// TwinCAT 3 PLC project x_template_xPlc
// Title: x_template_xPlc
// Company: TcOpen.MTS
// ProjectVersion: 0.6.0.913
// ProgramVersion: 3.1.4023.0
// libraries:
//   Tc2_Standard, * (Beckhoff Automation GmbH)
//   Tc2_System, * (Beckhoff Automation GmbH)
//   Tc3_Module, * (Beckhoff Automation GmbH)
//   TcoAbbRobotics, 0.11.0.74 (Vortex.Library)
//   TcoAbstractions, 0.11.0.74 (Vortex.Library)
//   TcoAimTtiPowerSupply, 0.11.0.74 (Vortex.Library)
//   TcoCognexVision, 0.11.0.74 (Vortex.Library)
//   TcoCore, 0.11.0.74 (Vortex.Library)
//   TcoData, 0.11.0.74 (Vortex.Library)
//   TcoDrivesBeckhoff, 0.11.0.74 (Vortex.Library)
//   TcoElements, 0.11.0.74 (Vortex.Library)
//   TcoInspectors, 0.11.0.74 (Vortex.Library)
//   TcoIo, 0.11.0.74 (Vortex.Library)
//   TcoKukaRobotics, 0.11.0.74 (Vortex.Library)
//   TcoMitsubishiRobotics, 0.11.0.74 (Vortex.Library)
//   TcoPneumatics, 0.11.0.74 (Vortex.Library)
//   TcoRexrothPress, 0.11.0.74 (Vortex.Library)
//   TcoTixonFeeding, 0.11.0.74 (Vortex.Library)
//   TcoUrRobotics, 0.11.0.74 (Vortex.Library)
//   TcoUtilities, 0.11.0.74 (Vortex.Library)
// project tree:
//   Abstractions/Components/ArrayRenderingExample/ SampleArrayToRender.TcDUT, SampleDataItem.TcDUT
//   Abstractions/Components/MtsFeeding/Blisters/Plb/ TcoPlbPaletizator.TcPOU, TcoPlbPaletizator_Components.TcDUT, TcoPlbPaletizator_Config_v_1_x_x.TcDUT, TcoPlbPaletizator_Control_v_1_x_x.TcDUT, TcoPlbPaletizator_Positions.TcPOU, TcoPlbPaletizator_Status_v_1_x_x.TcDUT
//   Abstractions/Components/MtsFeeding/Blisters/Plr/ TcoPlrPaletizator.TcPOU, TcoPlrPaletizator_Components.TcDUT, TcoPlrPaletizator_Config_v_1_x_x.TcDUT, TcoPlrPaletizator_Control_v_1_x_x.TcDUT, TcoPlrPaletizator_Status_v_1_x_x.TcDUT
//   Abstractions/Components/MtsFeeding/Blisters/Pls/ TcoPlsPaletizator.TcPOU, TcoPlsPaletizator_Components.TcDUT, TcoPlsPaletizator_Config_v_1_x_x.TcDUT, TcoPlsPaletizator_Control_v_1_x_x.TcDUT, TcoPlsPaletizator_Status_v_1_x_x.TcDUT
//   Abstractions/Components/MtsFeeding/Blisters/ TcoFeeding_Config_v_1_x_x.TcDUT, TcoFeeding_Status_v_1_x_x.TcDUT
//   Abstractions/Components/MtsFeeding/Components/OscilatingConveyorFeeder/ eTcoOscilatingConveyorOscilationModes.TcDUT, eTcoOscilatingConveyorStatus.TcDUT, TcoOscilatingConveyorFeeder.TcPOU, TcoOscilatingConveyorFeederComponents.TcDUT, TcoOscilatingConveyorFeeder_Config_v_1_x_x.TcDUT, TcoOscilatingConveyorFeeder_Control_v_1_x_x.TcDUT, TcoOscilatingConveyorFeeder_DesignerSpecificData.TcPOU, TcoOscilatingConveyorFeeder_PcToPlc.TcDUT, TcoOscilatingConveyorFeeder_PlcToPc.TcDUT, TcoOscilatingConveyorFeeder_Status_v_1_x_x.TcDUT
//   Abstractions/Components/MtsFeeding/ TcoFeedingSequenceTask.TcPOU
//   Abstractions/Components/Rework/ eReworkResults.TcDUT, ReworkData.TcDUT, ReworkInstructionTask.TcPOU
//   Abstractions/Components/TS/EqTransfer/ eTcoEq2TransferConfiguration.TcDUT, eTcoEq2TransferHandlingMode.TcDUT, TcoEq2Transfer.TcPOU, TcoEq2TransferComponents.TcDUT, TcoEq2Transfer_Config.TcDUT, TcoEq2Transfer_Control.TcDUT, TcoEq2Transfer_Status.TcDUT
//   Abstractions/Components/TS/RotaryTrabsferWithLift/ TcoLiftingRotaryTransfer.TcPOU, TcoLiftingRotaryTransferComponents.TcDUT, TcoLiftingRotaryTransfer_Config.TcDUT, TcoLiftingRotaryTransfer_Control.TcDUT, TcoLiftingRotaryTransfer_Status.TcDUT
//   Abstractions/Components/TS/RotaryTransfer/ TcoRotaryTransfer.TcPOU, TcoRotaryTransferComponents.TcDUT, TcoRotaryTransfer_Config.TcDUT, TcoRotaryTransfer_Control.TcDUT, TcoRotaryTransfer_Status.TcDUT
//   Abstractions/Components/TS/WorkPosition/ TcoTransferSystemComponent.TcPOU, TcoTransferSystemComponents.TcDUT, TcoTransferSystem_Config.TcDUT, TcoTransferSystem_Control.TcDUT, TcoTransferSystem_Status.TcDUT
//   Abstractions/Components/WrappedComponent/ WrappedComponentExample.TcPOU, WrappedComponentExample_Config.TcDUT, WrappedComponentExample_Control.TcDUT, WrappedComponentExample_Status.TcDUT, WrappedComponentsExample.TcDUT
//   Abstractions/CUBase/ CuBaseRecurringFail.TcDUT, CuBaseRecurringFailures.TcDUT, CUBase.TcPOU, CUBaseStatusInfo.TcDUT, CUBaseSettings.TcDUT, CUComponentsBase.TcDUT (not stored), ICUBase.TcIO, ICUTask.TcIO (not stored), OperatorInfo.TcDUT (not stored)
//   Abstractions/CUBase/Data/ BasicCounterData.TcDUT, CuHeader.TcDUT, CUProcessDataBase.TcDUT, CUTechnologicalDataBase.TcDUT, eCUMode.TcDUT (not stored), eCUState.TcDUT, eDataEntityInvokeType.TcDUT, EntityHeader.TcDUT
//   Abstractions/CUBase/RemoteTasks/ ProductionPlaner.TcPOU
//   Abstractions/CUBase/Tasks/ CUBaseAutomat.TcPOU, CUBaseSuspend.TcPOU, CUBaseGround.TcPOU (not stored), CUBaseRecover.TcPOU
//   Abstractions/Generic/LightTower/ TcoLightTower.TcPOU, TcoLightTower_Config.TcDUT, TcoLightTower_Info.TcDUT, TcoLightTower_Status.TcDUT
//   Abstractions/Generic/NotificationPanel/ NotificationPanel.TcPOU, NotificationPanelInfo.TcDUT
//   Abstractions/Generic/TagsPairing/ eTagPairingAnswer.TcDUT, eTagPairingMode.TcDUT, eTagPairingStatus.TcDUT, PairTagTask.TcPOU, TagsPairing.TcDUT
//   Abstractions/Safety/ControlButtons/ ITcoControlButtons.TcIO, TcoControlButtons.TcPOU, TcoControledZone_Info.TcDUT
//   Abstractions/Safety/ControlledZone/ TcoControlledZone.TcPOU, TcoControlledZoneActionTask.TcPOU, TcoControlledZone_Config.TcDUT, TcoControlledZone_Status.TcDUT
//   Abstractions/Safety/ControlVoltage/ ITcoControlVoltage.TcIO, TcoControlVoltage.TcPOU
//   Abstractions/Safety/DoorCircuit/ TcoDoorCircuit_Status.TcDUT, TcoDoorCircuit_Config.TcDUT, TcoDoorCircuit.TcPOU, ITcoDoorCircuit.TcIO
//   Abstractions/Safety/Doors/ ITcoDoorLock.TcIO (not stored), TcoStandardDoor.TcPOU, TcoBasicDoor.TcPOU
//   Abstractions/Safety/Estop/ TcoEmergencyStop.TcPOU
//   Abstractions/Safety/KeyMode/ TcoKeyMode_Config.TcDUT, TcoKeyMode_Status.TcDUT, TcoKeyMode.TcPOU, ITcoKeyMode.TcIO
//   Abstractions/Safety/KeyNormalService/ TcoKeyNormalService.TcPOU, ITcoKeyNormalSevice.TcIO
//   Abstractions/TcoCore/ CycleTimeAnalitics.TcDUT, TcoInnerTask.TcPOU (not stored), TcoTaskedSequencer.TcPOU, TcoTaskedService.TcPOU (not stored)
//   Abstractions/Technology/ eStations.TcDUT (not stored)
//   DUTs/IO_Specific/Aventics/ AES_D_BC_ECAT_Gen2_32bytes_Data_Inputs.TcDUT, AES_D_BC_ECAT_Gen2_32bytes_Data_Outputs.TcDUT, AES_D_BC_ECAT_Gen2_4bytes_Data_Inputs.TcDUT, AES_D_BC_ECAT_Gen2_4bytes_Data_Outputs.TcDUT
//   / MAIN.TcPOU (not stored), PlcTask.TcTTO
//   Technology/CU00x/Automat/ CU00xAutomatParalell_1_Task.TcPOU, CU00xAutomatTask.TcPOU
//   Technology/CU00x/Components/ CU00xExamplesOfComponents.TcDUT, CU00xComponents.TcDUT
//   Technology/CU00x/Data/ CU00xTechnologicalData.TcDUT, CU00xDialogContent.TcPOU, CU00xProcessData.TcDUT
//   Technology/CU00x/Ground/ CU00xGroundTask.TcPOU
//   Technology/CU00x/Manual/ CU00xManualTask.TcPOU
//   Technology/CU00x/Positions/ CU00xTestMultiPositions.TcPOU, Cu00xTestPositions.TcPOU
//   Technology/CU00x/Safety/Suspend/ CU00xSuspendTask.TcPOU
//   Technology/CU00x/Safety/Recover/ CU00xRecoverTask.TcPOU
//   Technology/Data/ InternalStorage.TcPOU, ProcessData.TcDUT, ProcessDataManager.TcPOU, TcoEntityBase.TcDUT, TechnologicalDataManager.TcPOU (not stored), TechnologyData.TcDUT
//   Technology/CU00x/ CU00x.TcPOU
//   Technology/ Technology.TcPOU, TechnologyComponents.TcDUT
//   DUTs/IO/PDOs/ Device_State_F0482DC3.TcDUT (not stored), Device_Control_6258066A.TcDUT (not stored), Inputs_23559BB0.TcDUT (not stored), Outputs_FC2FACAD.TcDUT (not stored), Modules_85784B27.TcDUT (not stored), Channel_830843C1.TcDUT, Channel_42CA91F7.TcDUT
//   DUTs/IO/Boxes/ EK1200_013D0B49.TcDUT, EK1122_1FC0878B.TcDUT, AES_510494FB.TcDUT (not stored), EPP1322_1FC0878B.TcDUT (not stored), EPP1809_32157CFD.TcDUT (not stored), EPP1008_78E8D3DD.TcDUT (not stored), EL1809_32157CFD.TcDUT, EL2809_2B6483BD.TcDUT, EL9011_D65D3D32.TcDUT
//   DUTs/IO/Devices/ SyncUnitTasks_4BE01469.TcDUT, SyncUnits_67D36DDA.TcDUT
//   DUTs/IO/Topology/ EK_E812B8FA.TcDUT (not stored), EC_4E5C738F.TcDUT (not stored), EC_245FBB9A.TcDUT (not stored)
//   GVLs/ GVL_iXlinker.TcGVL
// real-time tasks:
//   TASK PlcTask: cycle T#10ms, priority 20, ADS port 350
//   TASK PlcTask1: cycle T#10ms, priority 21, ADS port 351
// I/O:
//   DEVICE EC1 (disabled), AmsNetId 192.168.4.1.7.1
//     (EK1200) [EK1200-5000 EtherCAT Power supply (2A E-Bus)]
//       EC (EK1122) [EK1122 2 port EtherCAT junction]
//       PN (EL6631) [EL6631 PROFINET IO Controller]
//       IA1 (EL1809) [EL1809 16Ch. Dig. Input 24V, 3ms]
//       QA1 (EL2809) [EL2809 16Ch. Dig. Output 24V, 0.5A]
//       Term 6 (EL4004) [EL4004 4Ch. Ana. Output 0-10V, 12bit]
//       Term 7 (EL7342) [EL7342 2Ch. DC motor output stage (50V, 3.5A)]
//       Term 8 (EL4004) [EL4004 4Ch. Ana. Output 0-10V, 12bit]
//       Term 9 (EL6001) [EL6001 Interface (RS232)]
//       Term 13 (EL9011) [EL9011 End Terminal]
//   DEVICE EC (disabled), AmsNetId 192.168.4.1.2.1
//     EC [EK1200-5000 EtherCAT Power supply (2A E-Bus)]
//       EK [EK1122 2 port EtherCAT junction]
//         PNEU [AES Fieldbus Coupler Gen2]
//           modules: Modules
//         AB [EPP1322-0001 3 port EtherCAT P gateway]
//         AB21 [EPP1809-0021 16 Ch. Dig. Input 24V, 3ms, M8]
//         AB22 [EPP1809-0021 16 Ch. Dig. Input 24V, 3ms, M8]
//         AB23 [EPP1008-0001 8 Ch. Dig. Input 24V, 3ms, M8]
//         AB24 [EPP1008-0001 8 Ch. Dig. Input 24V, 3ms, M8]
//       IA1 [EL1809 16Ch. Dig. Input 24V, 3ms]
//       QA1 [EL2809-0015 16Ch. Dig. Output 24V DC, 0.35A, not short-circuit proof]
//       Term 11 (EL9011) [EL9011 End Terminal]
// variable links:
//   x_template_xPlc/x_template_xPlc Instance <-> EC
//     PlcTask Inputs/GVL_iXlinker.EC.InfoData.AmsNetId <-> InfoData/AmsNetId
//     PlcTask Inputs/GVL_iXlinker.EC.InfoData.CfgSlaveCount <-> InfoData/CfgSlaveCount
//     PlcTask Inputs/GVL_iXlinker.EC.InfoData.ChangeCount <-> InfoData/ChangeCount
//     PlcTask Inputs/GVL_iXlinker.EC.InfoData.DevId <-> InfoData/DevId
//     PlcTask Inputs/GVL_iXlinker.EC.Inputs.DevState <-> Inputs/DevState
//     PlcTask Inputs/GVL_iXlinker.EC.Inputs.Frm0InputToggle <-> Inputs/Frm0InputToggle
//     PlcTask Inputs/GVL_iXlinker.EC.Inputs.Frm0State <-> Inputs/Frm0State
//     PlcTask Inputs/GVL_iXlinker.EC.Inputs.Frm0WcState <-> Inputs/Frm0WcState
//     PlcTask Inputs/GVL_iXlinker.EC.Inputs.SlaveCount <-> Inputs/SlaveCount
//     PlcTask Inputs/GVL_iXlinker.EC.SyncUnits._default.PlcTask.InfoData.ObjectId <-> SyncUnits/<default>/PlcTask/InfoData/ObjectId
//     PlcTask Inputs/GVL_iXlinker.EC.SyncUnits._default.PlcTask.InfoData.SlaveCount <-> SyncUnits/<default>/PlcTask/InfoData/SlaveCount
//     PlcTask Inputs/GVL_iXlinker.EC.SyncUnits._default.PlcTask.InfoData.State <-> SyncUnits/<default>/PlcTask/InfoData/State
//     PlcTask Inputs/GVL_iXlinker.EC.SyncUnits._default.PlcTask.WcState.WcState <-> SyncUnits/<default>/PlcTask/WcState/WcState
//     PlcTask Outputs/GVL_iXlinker.EC.Outputs.DevCtrl <-> Outputs/DevCtrl
//     PlcTask Outputs/GVL_iXlinker.EC.Outputs.Frm0Ctrl <-> Outputs/Frm0Ctrl
//     PlcTask Outputs/GVL_iXlinker.EC.Outputs.Frm0WcCtrl <-> Outputs/Frm0WcCtrl
//   x_template_xPlc/x_template_xPlc Instance <-> EC/EC/EK
//     PlcTask Inputs/GVL_iXlinker.EC.EC.EK.InfoData.State <-> InfoData/State
//   x_template_xPlc/x_template_xPlc Instance <-> EC/EC/EK/AB
//     PlcTask Inputs/GVL_iXlinker.EC.EC.EK.AB.InfoData.State <-> InfoData/State
//   x_template_xPlc/x_template_xPlc Instance <-> EC/EC/EK/AB21
//     PlcTask Inputs/GVL_iXlinker.EC.EC.EK.AB21.Channel_{1..16}.Input <-> Channel {1..16}/Input  (16 links)
//     PlcTask Inputs/GVL_iXlinker.EC.EC.EK.AB21.InfoData.State <-> InfoData/State
//     PlcTask Inputs/GVL_iXlinker.EC.EC.EK.AB21.WcState.InputToggle <-> WcState/InputToggle
//     PlcTask Inputs/GVL_iXlinker.EC.EC.EK.AB21.WcState.WcState <-> WcState/WcState
//   x_template_xPlc/x_template_xPlc Instance <-> EC/EC/EK/AB22
//     PlcTask Inputs/GVL_iXlinker.EC.EC.EK.AB22.Channel_{1..16}.Input <-> Channel {1..16}/Input  (16 links)
//     PlcTask Inputs/GVL_iXlinker.EC.EC.EK.AB22.InfoData.State <-> InfoData/State
//     PlcTask Inputs/GVL_iXlinker.EC.EC.EK.AB22.WcState.InputToggle <-> WcState/InputToggle
//     PlcTask Inputs/GVL_iXlinker.EC.EC.EK.AB22.WcState.WcState <-> WcState/WcState
//   x_template_xPlc/x_template_xPlc Instance <-> EC/EC/EK/AB23
//     PlcTask Inputs/GVL_iXlinker.EC.EC.EK.AB23.Channel_{1..8}.Input <-> Channel {1..8}/Input  (8 links)
//     PlcTask Inputs/GVL_iXlinker.EC.EC.EK.AB23.InfoData.State <-> InfoData/State
//     PlcTask Inputs/GVL_iXlinker.EC.EC.EK.AB23.WcState.InputToggle <-> WcState/InputToggle
//     PlcTask Inputs/GVL_iXlinker.EC.EC.EK.AB23.WcState.WcState <-> WcState/WcState
//   x_template_xPlc/x_template_xPlc Instance <-> EC/EC/EK/AB24
//     PlcTask Inputs/GVL_iXlinker.EC.EC.EK.AB24.Channel_{1..8}.Input <-> Channel {1..8}/Input  (8 links)
//     PlcTask Inputs/GVL_iXlinker.EC.EC.EK.AB24.InfoData.State <-> InfoData/State
//     PlcTask Inputs/GVL_iXlinker.EC.EC.EK.AB24.WcState.InputToggle <-> WcState/InputToggle
//     PlcTask Inputs/GVL_iXlinker.EC.EC.EK.AB24.WcState.WcState <-> WcState/WcState
//   x_template_xPlc/x_template_xPlc Instance <-> EC/EC/EK/PNEU
//     PlcTask Inputs/GVL_iXlinker.EC.EC.EK.PNEU.Device_State.CommonValve <-> Device_State/CommonValve
//     PlcTask Inputs/GVL_iXlinker.EC.EC.EK.PNEU.Device_State.Configuration_Error_IO_Module <-> Device_State/Configuration Error IO-Module
//     PlcTask Inputs/GVL_iXlinker.EC.EC.EK.PNEU.Device_State.Configuration_Error_Valve <-> Device_State/Configuration Error Valve
//     PlcTask Inputs/GVL_iXlinker.EC.EC.EK.PNEU.Device_State.Configuratipn_Error_SLS <-> Device_State/Configuratipn Error SLS
//     PlcTask Inputs/GVL_iXlinker.EC.EC.EK.PNEU.Device_State.Count_IO_Module_to_big <-> Device_State/Count IO-Module to big
//     PlcTask Inputs/GVL_iXlinker.EC.EC.EK.PNEU.Device_State.Heardbeat_x <-> Device_State/Heardbeat
//     PlcTask Inputs/GVL_iXlinker.EC.EC.EK.PNEU.Device_State.IO_1_8 <-> Device_State/IO:1-8
//     PlcTask Inputs/GVL_iXlinker.EC.EC.EK.PNEU.Device_State.IO_9_10 <-> Device_State/IO:9-10
//     PlcTask Inputs/GVL_iXlinker.EC.EC.EK.PNEU.Device_State.Switchcounter_Error <-> Device_State/Switchcounter Error
//     PlcTask Inputs/GVL_iXlinker.EC.EC.EK.PNEU.Device_State.UA_OFF <-> Device_State/UA OFF
//     PlcTask Inputs/GVL_iXlinker.EC.EC.EK.PNEU.Device_State.UL_OFF <-> Device_State/UL OFF
//     PlcTask Inputs/GVL_iXlinker.EC.EC.EK.PNEU.Device_State.Undervoltage_5V <-> Device_State/Undervoltage 5V
//     PlcTask Inputs/GVL_iXlinker.EC.EC.EK.PNEU.Device_State.Undervoltage_UA <-> Device_State/Undervoltage UA
//     PlcTask Inputs/GVL_iXlinker.EC.EC.EK.PNEU.Device_State.Undervoltage_UL <-> Device_State/Undervoltage UL
//     PlcTask Inputs/GVL_iXlinker.EC.EC.EK.PNEU.Device_State.Unknown_Module_ID <-> Device_State/Unknown Module ID
//     PlcTask Inputs/GVL_iXlinker.EC.EC.EK.PNEU.Device_State.ValveExtSupplyDiag_1_6 <-> Device_State/ValveExtSupplyDiag:1-6
//     PlcTask Inputs/GVL_iXlinker.EC.EC.EK.PNEU.InfoData.AdsAddr <-> InfoData/AdsAddr
//     PlcTask Inputs/GVL_iXlinker.EC.EC.EK.PNEU.InfoData.State <-> InfoData/State
//     PlcTask Inputs/GVL_iXlinker.EC.EC.EK.PNEU.Modules.Inputs.digital_Data_I[{0..31}] <-> Modules/Inputs/digital Data I_{0..31}  (32 links)
//     PlcTask Inputs/GVL_iXlinker.EC.EC.EK.PNEU.WcState.InputToggle <-> WcState/InputToggle
//     PlcTask Inputs/GVL_iXlinker.EC.EC.EK.PNEU.WcState.WcState <-> WcState/WcState
//     PlcTask Outputs/GVL_iXlinker.EC.EC.EK.PNEU.Device_Control.Default_Modul_Control <-> Device_Control/Default_Modul_Control
//     PlcTask Outputs/GVL_iXlinker.EC.EC.EK.PNEU.Device_Control.Freeze_Output <-> Device_Control/Freeze Output
//     PlcTask Outputs/GVL_iXlinker.EC.EC.EK.PNEU.Device_Control.HL_Swap <-> Device_Control/HL_Swap
//     PlcTask Outputs/GVL_iXlinker.EC.EC.EK.PNEU.Device_Control.Web_App_Disable <-> Device_Control/Web App Disable
//     PlcTask Outputs/GVL_iXlinker.EC.EC.EK.PNEU.Modules.Outputs.digital_Data_O[{0..31}] <-> Modules/Outputs/digital Data O_{0..31}  (32 links)
//   x_template_xPlc/x_template_xPlc Instance <-> EC/EC/IA1
//     PlcTask Inputs/GVL_iXlinker.EC.EC.IA1.Channel_{1..16}.Input <-> Channel {1..16}/Input  (16 links)
//     PlcTask Inputs/GVL_iXlinker.EC.EC.IA1.InfoData.State <-> InfoData/State
//     PlcTask Inputs/GVL_iXlinker.EC.EC.IA1.WcState.InputToggle <-> WcState/InputToggle
//     PlcTask Inputs/GVL_iXlinker.EC.EC.IA1.WcState.WcState <-> WcState/WcState
//   x_template_xPlc/x_template_xPlc Instance <-> EC/EC/QA1
//     PlcTask Inputs/GVL_iXlinker.EC.EC.QA1.InfoData.State <-> InfoData/State
//     PlcTask Inputs/GVL_iXlinker.EC.EC.QA1.WcState.WcState <-> WcState/WcState
//     PlcTask Outputs/GVL_iXlinker.EC.EC.QA1.Channel_{1..16}.Output <-> Channel {1..16}/Output  (16 links)

CONFIGURATION x_template_xPlc
    RESOURCE PLC ON TwinCAT3
        TASK PlcTask(INTERVAL := T#4ms, PRIORITY := 20);
        PROGRAM MAIN WITH PlcTask : MAIN;
    END_RESOURCE
END_CONFIGURATION

// ---- Abstractions/Components/ArrayRenderingExample/SampleArrayToRender.TcDUT
TYPE SampleArrayToRender :
STRUCT
	Data	:	ARRAY  [0..100] OF SampleDataItem;
END_STRUCT
END_TYPE

// ---- Abstractions/Components/ArrayRenderingExample/SampleDataItem.TcDUT
TYPE SampleDataItem :
STRUCT
 	Measured : BOOL;
    Overrided : BOOL;
    Marginal : BOOL;
    FinalResults : BOOL;
END_STRUCT
END_TYPE

// ---- Abstractions/Components/MtsFeeding/Blisters/Plb/TcoPlbPaletizator_Components.TcDUT
TYPE TcoPlbPaletizator_Components EXTENDS TcoCore.TcoStruct:
STRUCT
	
	{attribute wpf [Container(Layout.Stack)]}
	{attribute addProperty Name "<#(I1) Zasobnik blistrov 1 Nema minimalne mnozstvo#>"}
	I1_iBuffer1HasNotCriticalLevel : TcoElements.TcoDi(THISSTRUCT);

	{attribute addProperty Name "<#(I2) Zasobnik blistrov 1 kus pripraveny na odoberanie#>"}
	I2_iBuffer1IsReadyToLoad : TcoElements.TcoDi(THISSTRUCT);
	
	{attribute addProperty Name "<#(I3) Zasobnik blistrov 2 Nema minimalne mnozstvo#>"}
	I3_iBuffer2HasNotCriticalLevel : TcoElements.TcoDi(THISSTRUCT);


	{attribute addProperty Name "<#(I4) Zasobnik blistrov 2 kus pripraveny na odoberanie#>"}
	I4_iBuffer2IsReadyToLoad : TcoElements.TcoDi(THISSTRUCT);
	
	{attribute addProperty Name "<#(I5) Zasobnik blistrov 3 Nema minimalne mnozstvo#>"}
	I5_iBuffer3HasNotCriticalLevel : TcoElements.TcoDi(THISSTRUCT);
	
	{attribute addProperty Name "<#(I6) Zasobnik blistrov 3 kus pripraveny na odoberanie#>"}
	I6_iBuffer3IsReadyToLoad : TcoElements.TcoDi(THISSTRUCT);
	
	{attribute addProperty Name "<#(I7) Zasobnik blistrov 4 Nema minimalne mnozstvo#>"}
	I7_iBuffer4HasNotCriticalLevel : TcoElements.TcoDi(THISSTRUCT);
	
	{attribute addProperty Name "<#(I8) Zasobnik blistrov 4 kus pripraveny na odoberanie#>"}
	I8_iBuffer4IsReadyToLoad : TcoElements.TcoDi(THISSTRUCT);
	
	{attribute addProperty Name "<#(I9) Zasobnik prazdnych blistrov 1 plny#>"}
	I9_iThrowBuffer1Isfull : TcoElements.TcoDi(THISSTRUCT);
	
	{attribute addProperty Name "<#(I10)Zasobnik prazdnych blistrov 2 plny#>"}
	I10_iThrowBuffer2Isfull : TcoElements.TcoDi(THISSTRUCT);
	
	{attribute addProperty Name "<#(I11) Blister v pracovnej pozicii#>"}
	I11_BlisterInWorkPosition : TcoElements.TcoDi(THISSTRUCT);
	
	{attribute addProperty Name "<#(I12) Blister uchopeny spravne(volitelny)#>"}
	I12_BlisterPickedCorrectly : TcoElements.TcoDi(THISSTRUCT);
	
	{attribute wpf [Container(Layout.Stack)]}
	{attribute addProperty Name "<#(P1)Pozicna jednoka#>"}
	P1_PositionUnit :TcoPneumatics.TcoCylinder(THISSTRUCT);
	{attribute addProperty Name "<#(P2)Upevnenie blistra#>"}
	P2_FixUnit :TcoPneumatics.TcoDoubleCylinder(THISSTRUCT);
	
	{attribute wpf [Container(Layout.Stack)]}
	{attribute addProperty Name "<#Manipulator#>"}
	Manipulator :TcoDrivesBeckhoff.TcoSingleAxis(THISSTRUCT);
	
	{attribute wpf [Container(Layout.Stack,"Vseobecne")]}
	
	{attribute addProperty Name "(Q1) <#Signalizacia upozornenia R#>"}
	Q1_AttentionSignalisationR : TcoElements.TcoDo(THISSTRUCT);
	{attribute addProperty Name "(Q2) <#Signalizacia upozornenia G#>"}
	Q2_AttentionSignalisationG : TcoElements.TcoDo(THISSTRUCT);
	{attribute addProperty Name "(Q3) <#Signalizacia upozornenia B#>"}
	Q3_AttentionSignalisationB : TcoElements.TcoDo(THISSTRUCT);

	
	
END_STRUCT
END_TYPE

// ---- Abstractions/Components/MtsFeeding/Blisters/Plb/TcoPlbPaletizator_Config_v_1_x_x.TcDUT
TYPE
    TcoPlbPaletizator_Config_v_1_x_x EXTENDS  TcoFeeding_Config_v_1_x_x:
    STRUCT

      

        {attribute addProperty Name "<#Manipulator - Pozicie nazov #>"}
        PositionsSetName : STRING;

        {attribute addProperty Name "<#Zasobnik 1 zakazany#>"}
        Buffer1Disabled : BOOL;

        {attribute addProperty Name "<#Zasobnik 2 zakazany#>"}
        Buffer2Disabled : BOOL;

        {attribute addProperty Name "<#Zasobnik 2 zakazany#>"}
        Buffer3Disabled : BOOL;

        {attribute addProperty Name "<#Zasobnik 2 zakazany#>"}
        Buffer4Disabled : BOOL;

        {attribute addProperty Name "<#Zasobnik prazdnych 1 zakazany#>"}
        EmptyBuffer1Disabled : BOOL;

        {attribute addProperty Name "<#Zasobnik prazdnych 2 zakazany#>"}
        EmptyBuffer2Disabled : BOOL;
    END_STRUCT
END_TYPE

// ---- Abstractions/Components/MtsFeeding/Blisters/Plb/TcoPlbPaletizator_Control_v_1_x_x.TcDUT
TYPE TcoPlbPaletizator_Control_v_1_x_x EXTENDS TcoCore.TcoStruct:
STRUCT

		ResetOnlyManipulator: BOOL;
		
END_STRUCT
END_TYPE

// ---- Abstractions/Components/MtsFeeding/Blisters/Plb/TcoPlbPaletizator_Status_v_1_x_x.TcDUT
TYPE
    TcoPlbPaletizator_Status_v_1_x_x EXTENDS TcoFeeding_Status_v_1_x_x:
    STRUCT


        ReadyToUnloadComponents : BOOL;
        OutBufferFull : BOOL;
		EntryBufferEmpty : BOOL;
    END_STRUCT
END_TYPE

// ---- Abstractions/Components/MtsFeeding/Blisters/Plr/TcoPlrPaletizator_Components.TcDUT
TYPE
    TcoPlrPaletizator_Components EXTENDS TcoCore.TcoStruct :
    STRUCT

        {attribute wpf [Container(Layout.Stack,"Vstup Blistrov")]}
        {attribute addProperty Name "<#(I1) Pritomnost blistra na vstupnej zarazke 1 - vstup#>"}
        I1_PresentBlisterAtEntryStopper1 : TcoElements.TcoDi(THISSTRUCT);

        {attribute addProperty Name "<#(I2) Pritomnost blistra na vstupnej zarazke 1 - plny(WIPA)#>"}
        I2_PresentBlisterAtEntryStopper1Wipa : TcoElements.TcoDi(THISSTRUCT);

        {attribute addProperty Name "<#(I3) Spravnost nalozenia blistra na vstupnej zarazke 1 - vstup#>"}
        I3_NotLoadedCorrectlyAtEntryStopper1 : TcoElements.TcoDi(THISSTRUCT);

        {attribute addProperty Name "<#(I4) Pritomnost blistra na vstupnej zarazke 2 - vstup#>"}
        I4_PresentBlisterAtEntryStopper2 : TcoElements.TcoDi(THISSTRUCT);

        {attribute addProperty Name "<#(I6) Pritomnost blistra na vstupnej zarazke 2 - plny(WIPA)#>"}
        I5_PresentBlisterAtEntryStopper2Wipa : TcoElements.TcoDi(THISSTRUCT);

        {attribute addProperty Name "<#(I6) Pritomnost blistra na vstupnej zarazke 3 - vstup#>"}
        I6_PresentBlisterAtEntryStopper3 : TcoElements.TcoDi(THISSTRUCT);

        {attribute addProperty Name "<#(I7) Pritomnost blistra na vstupnej zarazke 3 - plny(WIPA)#>"}
        I7_PresentBlisterAtEntryStopper3Wipa : TcoElements.TcoDi(THISSTRUCT);

        {attribute addProperty Name "<#(I8) Pritomnost blistra na vstupnej zarazke 4 - vstup#>"}
        I8_PresentBlisterAtEntryStopper4 : TcoElements.TcoDi(THISSTRUCT);

        {attribute addProperty Name "<#(I9) Pritomnost blistra na vstupnej zarazke 4 - plny(WIPA)#>"}
        I9_PresentBlisterAtEntryStopper4Wipa : TcoElements.TcoDi(THISSTRUCT);

        {attribute addProperty Name "<#(Q4)Vstupny dopravnik#>"}
        Q4_EntryConvRun : TcoElements.TcoDo(THISSTRUCT);

        {attribute addProperty Name "<#Vstupny dopravnik reverz#>"}
        Q5_EntryConvRunReverse : TcoElements.TcoDo(THISSTRUCT);

        {attribute addProperty Name "<#(PR1)(PR1.1) Zarazka Vstupny dopravnik#>"}
        PR1_StopperConveyorEntry1 : TcoPneumatics.TcoDoubleCylinder(THISSTRUCT);

        {attribute addProperty Name "<#(PR2)(PR2.1) Zarazka Vstupny dopravnik#>"}
        PR2_StopperConveyorEntry2 : TcoPneumatics.TcoDoubleCylinder(THISSTRUCT);

        {attribute addProperty Name "<#(PR3)(PR3.1) Zarazka Vstupny dopravnik#>"}
        PR3_StopperConveyorEntry3 : TcoPneumatics.TcoDoubleCylinder(THISSTRUCT);

        {attribute addProperty Name "<#(PR4)(PR4.1) Zarazka Vstupny dopravnik#>"}
        PR4_StopperConveyorEntry4 : TcoPneumatics.TcoDoubleCylinder(THISSTRUCT);

        {attribute addProperty Name "<#(PR5)(PR5.1) Zarazka Vystupny dopravnik#>"}
        PR5_StopperConveyorOutgoing1 : TcoPneumatics.TcoDoubleCylinder(THISSTRUCT);

		
        {attribute addProperty Name "<#(PR6)(PR6.1) Horizontalny prisun vstupnych blistrov#>"}
        PR6_HorizontalSepareEntyBlisters : TcoPneumatics.TcoDoubleCylinder(THISSTRUCT);

        {attribute addProperty Name "<#(PR7)(PR7.1) Horizontalny prisun vystupnych blistrov#>"}
        PR7_HorizontalSepareOutgoingBlisters : TcoPneumatics.TcoDoubleCylinder(THISSTRUCT);

        {attribute addProperty Name "<#(PR8) Vertikalne separovanie vstupnych blistrov 1#>"}
        PR8_VerticalSepareEntryBlister1 : TcoPneumatics.TcoCylinder(THISSTRUCT);

        {attribute addProperty Name "<#(PR9) Vertikalne separovanie vstupnych blistrov 2#>"}
        PR9_VerticalSepareEntryBlister2 : TcoPneumatics.TcoCylinder(THISSTRUCT);

        {attribute addProperty Name "<#(PR12)(PR12.1) Fixovanie vstupneho blistra z boku#>"}
        PR12_HorizontalHoldEntryBlister : TcoPneumatics.TcoDoubleCylinder(THISSTRUCT);

        {attribute wpf [Container(Layout.Stack,"Vystup Blistrov")]}
        {attribute addProperty Name "<#(I10) Pritomnost blistra na vystupnej zarazke 1 - vstup#>"}
        I10_PresentBlisterAtOutgoingStopper1 : TcoElements.TcoDi(THISSTRUCT);

        {attribute addProperty Name "<#(I11)Pritomnost blistra na vystupnej zarazke 1 - plny(WIPA)#>"}
        I11_PresentBlisterAtOutgoingStopper1Wipa : TcoElements.TcoDi(THISSTRUCT);

        {attribute addProperty Name "<#(I12) Vystupny zasobnik blistrov plny #>"}
        I12_OutgoingBufferIsFull : TcoElements.TcoDi(THISSTRUCT);
        {attribute addProperty Name "<#(I13)Vystupny dopravnik blistrov plny #>"}
        I13_OutgoingConveyorIsFull : TcoElements.TcoDi(THISSTRUCT);

        {attribute addProperty Name "<#(Q6) Vystupny dopravnik#>"}
        Q6_OutgoingConvRun : TcoElements.TcoDo(THISSTRUCT);

        {attribute addProperty Name "<#(Q7) Vystupny dopravnik reverz#>"}
        Q7_OutgoingConvRunReverse : TcoElements.TcoDo(THISSTRUCT);

        {attribute addProperty Name "<#(PR10) Vertikalne separovanie vstupnych blistrov 1#>"}
        PR10_VerticalSepareOutgoingBlister1 : TcoPneumatics.TcoCylinder(THISSTRUCT);

        {attribute addProperty Name "<#(PR11)Vertikalne separovanie vstupnych blistrov 2#>"}
        PR11_VerticalSepareOutgoingBlister2 : TcoPneumatics.TcoCylinder(THISSTRUCT);

		
		
        {attribute wpf [Container(Layout.Stack,"Vytah")]}
        {attribute addProperty Name "<#(I16) Pritomnost blistra v na vytahu - koniec #>"}
        I14_PresentBlisterInLiftEnd : TcoElements.TcoDi(THISSTRUCT);

        {attribute addProperty Name "<#(I15) Pritomnost blistra vo vytahu - vstup #>"}
        I15_PresentBlisterInLiftEntry : TcoElements.TcoDi(THISSTRUCT);

        {attribute addProperty Name "<#(Q8) Vytah dopravnik#>"}
        Q8_LiftConvRun : TcoElements.TcoDo(THISSTRUCT);

        {attribute addProperty Name "<#(Q9) Vytah dopravnik reverz#>"}
        Q9_LiftConvRunReverse : TcoElements.TcoDo(THISSTRUCT);

        {attribute addProperty Name "<#(PR13) Centrovanie blistra #>"}
        PR13_CenteringBlisterInLift : TcoPneumatics.TcoDoubleCylinder(THISSTRUCT);

        {attribute addProperty Name "<#(PR14) Vytah#>"}
        PR14_Lift : TcoPneumatics.TcoCylinder(THISSTRUCT);

        {attribute wpf [Container(Layout.Stack,"Vseobecne")]}
        {attribute addProperty Name "<#(I16)Tlacidlo - odoslanie blistrov#>"}
        I16_SendButton : TcoElements.TcoDi(THISSTRUCT);

        {attribute addProperty Name "<#(I17) Tlacidlo - privolanie blistrov(DOLE)#>"}
        I17_EmptyButton : TcoElements.TcoDi(THISSTRUCT);
		
		{attribute addProperty Name "<#(I18)Tlacidlo - privolanie blistrov(HORE)#>"}
		I18_EmptyKey : TcoElements.TcoDi(THISSTRUCT);	

        {attribute wpf [Container(Layout.Stack,"Vseobecne")]}

        {attribute addProperty Name "(Q1) <#Signalizacia upozornenia R#>"}
        Q1_AttentionSignalisationR : TcoElements.TcoDo(THISSTRUCT);
        {attribute addProperty Name "(Q2) <#Signalizacia upozornenia G#>"}
        Q2_AttentionSignalisationG : TcoElements.TcoDo(THISSTRUCT);
        {attribute addProperty Name "(Q3) <#Signalizacia upozornenia B#>"}
        Q3_AttentionSignalisationB : TcoElements.TcoDo(THISSTRUCT);

    END_STRUCT
END_TYPE

// ---- Abstractions/Components/MtsFeeding/Blisters/Plr/TcoPlrPaletizator_Config_v_1_x_x.TcDUT
TYPE
    TcoPlrPaletizator_Config_v_1_x_x EXTENDS TcoFeeding_Config_v_1_x_x :
    STRUCT
		
	{attribute addProperty Name "<#Vstupna zarazka (PR2) neaktivna#>"}
	PR2_StopperConveyorEntry2Disabled : BOOL;
	
	{attribute addProperty Name "<#Pridrziavanie blistra (PR12) neaktivne#>"}
	PR12_HorizontalHoldEntryBlisterDisabled:BOOL;
	
	{attribute addProperty Name "<#Automaticke stahovanie zarazky PR5 neaktivne#>"}
	UseAutoHidePr5Dispabled:BOOL;
	
	{attribute addProperty Name "<#Cas behu vstupneho dopravnika#>"}
	ConveyorEntryRunTime:TIME;
	
	{attribute addProperty Name "<#Cas behu vytupneho dopravnika#>"}
	ConveyorOutRunTime:TIME;

    END_STRUCT
END_TYPE

// ---- Abstractions/Components/MtsFeeding/Blisters/Plr/TcoPlrPaletizator_Control_v_1_x_x.TcDUT
TYPE TcoPlrPaletizator_Control_v_1_x_x EXTENDS TcoCore.TcoStruct:
STRUCT

		
END_STRUCT
END_TYPE

// ---- Abstractions/Components/MtsFeeding/Blisters/Plr/TcoPlrPaletizator_Status_v_1_x_x.TcDUT
TYPE
    TcoPlrPaletizator_Status_v_1_x_x EXTENDS TcoFeeding_Status_v_1_x_x:
    STRUCT

        
		EntryBufferEmpty:BOOL;
        BlisterReady : BOOL;
        OutBufferFull : BOOL;
    END_STRUCT
END_TYPE

// ---- Abstractions/Components/MtsFeeding/Blisters/Pls/TcoPlsPaletizator_Components.TcDUT
TYPE TcoPlsPaletizator_Components EXTENDS TcoCore.TcoStruct:
STRUCT
	
	{attribute wpf [Container(Layout.Stack)]}
	{attribute addProperty Name "(I1) <#Pritomnost blistra v presuvaci#>"}
	I1_PresentBlisterEntry : TcoElements.TcoDi(THISSTRUCT);
	
	{attribute addProperty Name "(I2) <#Pritomnost medzery medzi blistrami#>"}
	I2_PresentBlisterEntryEmptySpace : TcoElements.TcoDi(THISSTRUCT);
	
	{attribute addProperty Name "(I3) <#Zasobik blistrov prazdny#>"}
	I3_PresentBlistersInBufferEmpty : TcoElements.TcoDi(THISSTRUCT);

	
	{attribute addProperty Name "(I4) <#Pritomnost blistra v pracovnej pozicii#>"}
	I4_PresentBlisterInWorkingPos : TcoElements.TcoDi(THISSTRUCT);
		
	{attribute addProperty Name "(I5) <#Vystupny blister neje v sklzovom dopravniku#>"}
	I5_OutBlistersIsThrowedCorrectly : TcoElements.TcoDi(THISSTRUCT);
	
	{attribute addProperty Name "(I6) <#Vystupny blister snimanie vo vytahu#>"}
	I6_OutBlistersLisftSignal : TcoElements.TcoDi(THISSTRUCT);
	
	{attribute addProperty Name "(I7) <#Vystupny blister je nad Bufferom#>"}
	I7_OutBlistersIsAboveOutBuffer : TcoElements.TcoDi(THISSTRUCT);
	
	{attribute addProperty Name "(I8) <#Vystupny zasobnik je plny#>"}
	I8_OutBlistersBufferIsFull : TcoElements.TcoDi(THISSTRUCT);
	
	
	{attribute wpf [Container(Layout.Stack)]}
	{attribute addProperty Name "(P1) <#Vertikalny prisun vstupnych blistrov#>"}
	P1_VerticalSepareEntryBlisters : TcoPneumatics.TcoCylinder(THISSTRUCT);
	
	{attribute addProperty Name "(P2) <#Vertikalny prisun vstupnych blistrov #>"}
	P2_VerticalSepareEntryBlisters : TcoPneumatics.TcoCylinder(THISSTRUCT);
	
	{attribute addProperty Name "(P3) (P3.1) <#Horizontalny prisun vstupnych blistrov#>"}
	P3_HorizontalSepareEntryBlisters : TcoPneumatics.TcoDoubleCylinder(THISSTRUCT);
		
	{attribute addProperty Name "(P4) <#Prisun vstupneho blistra#>"}
	P4_FeedEntryBlister :TcoPneumatics.TcoCylinder(THISSTRUCT);
	
	{attribute addProperty Name "(P5) (P5.1)<#Horizontalny prisun vystupnych blistrov#>"}
	P5_HorizontalSepareOutBlisters : TcoPneumatics.TcoDoubleCylinder(THISSTRUCT);
	
	{attribute addProperty Name "(P6)<#Vertikalny prisun vystupnych blistrov#>"}
	P6_VerticalSepareOutBlister : TcoPneumatics.TcoCylinder(THISSTRUCT);
	
	{attribute addProperty Name "(P7) <#Podopretie vstupneho blistra#>"}
	P7_SupportEntryBlister : TcoPneumatics.TcoCylinder(THISSTRUCT);
	
	{attribute addProperty Name "(P8) (P8.1) <#Upevnenie zboku vstupneho blistra#>"}
	P8_FixEntryBlisterSide : TcoPneumatics.TcoDoubleCylinder(THISSTRUCT);
	
	{attribute addProperty Name "(P9) (P9.1) <#Zamknutue zhora vstupneho blistra#>"}
	P9_LockEntryBlisterTop : TcoPneumatics.TcoDoubleCylinder(THISSTRUCT);
	
	{attribute addProperty Name "(P10) (P10.1)<#Odelovac blistrov na vstupe#>"}
	P10_HoldEntrySepareOutBlister : TcoPneumatics.TcoDoubleCylinder(THISSTRUCT);
	
	
	
	{attribute wpf [Container(Layout.Stack,"Vseobecne")]}
	
	{attribute addProperty Name "(Q1) <#Signalizacia upozornenia R#>"}
	Q1_AttentionSignalisationR : TcoElements.TcoDo(THISSTRUCT);
	{attribute addProperty Name "(Q2) <#Signalizacia upozornenia G#>"}
	Q2_AttentionSignalisationG : TcoElements.TcoDo(THISSTRUCT);
	{attribute addProperty Name "(Q3) <#Signalizacia upozornenia B#>"}
	Q3_AttentionSignalisationB : TcoElements.TcoDo(THISSTRUCT);

	
	
END_STRUCT
END_TYPE

// ---- Abstractions/Components/MtsFeeding/Blisters/Pls/TcoPlsPaletizator_Config_v_1_x_x.TcDUT
TYPE
    TcoPlsPaletizator_Config_v_1_x_x EXTENDS TcoFeeding_Config_v_1_x_x :
    STRUCT

		
		
        {attribute addProperty Name "<#Zamykanie blistra zhora neaktive (P9)(P9.1)je nepritomne#>"}
		LockBlisterInPickPosInactive : BOOL;
		
		{attribute addProperty Name "<#Oddelovanie blistrov na vstupe neaktive (P10)(P10.1)je nepritomne#>"}
		SepareBlistersAtEntryInactive : BOOL;

    END_STRUCT
END_TYPE

// ---- Abstractions/Components/MtsFeeding/Blisters/Pls/TcoPlsPaletizator_Control_v_1_x_x.TcDUT
TYPE TcoPlsPaletizator_Control_v_1_x_x EXTENDS TcoCore.TcoStruct:
STRUCT

		
END_STRUCT
END_TYPE

// ---- Abstractions/Components/MtsFeeding/Blisters/Pls/TcoPlsPaletizator_Status_v_1_x_x.TcDUT
TYPE
    TcoPlsPaletizator_Status_v_1_x_x EXTENDS TcoFeeding_Status_v_1_x_x:
    STRUCT

        
		EntryBufferEmpty:BOOL;
        BlisterReady : BOOL;
        OutBufferFull : BOOL;
    END_STRUCT
END_TYPE

// ---- Abstractions/Components/MtsFeeding/Blisters/TcoFeeding_Config_v_1_x_x.TcDUT
TYPE
    TcoFeeding_Config_v_1_x_x EXTENDS TcoCore.TcoStruct :
    STRUCT

        InfoTime : TIME := T#5S;
        ErrorTime : TIME := T#0S;
        {attribute addProperty Name "<#Stabilizacny cas#>"}
        StabilisationTime : TIME := T#500MS;
        {attribute addProperty Name "<#Blink period#> "}
        BlinkTime : TIME := T#500MS;

        {attribute addProperty Name "<#Time to dissable safety#> "}
        TimeToDisableSafety : TIME := T#10S;

        {attribute addProperty Name "<#Volba krokoveho/Cyklickeho modu ovladna z vonka (SetSequencesToStep)#>"}
        StepModeManagableFromOutside : BOOL;

    END_STRUCT
END_TYPE

// ---- Abstractions/Components/MtsFeeding/Blisters/TcoFeeding_Status_v_1_x_x.TcDUT
TYPE
    TcoFeeding_Status_v_1_x_x EXTENDS TcoCore.TcoStruct :
    STRUCT

        ActionDescription : STRING;
        SafeCondition : BOOL;

    END_STRUCT
END_TYPE

// ---- Abstractions/Components/MtsFeeding/Components/OscilatingConveyorFeeder/eTcoOscilatingConveyorOscilationModes.TcDUT
{attribute 'qualified_only'}
{attribute 'strict'}
TYPE eTcoOscilatingConveyorOscilationModes :
(
	All:=0,
	Left:=1,
	Right:=2,
	Middle:=3,
	LeftRight:=4,
	LeftToRight := 5,
	RightToLeft :=6
);
END_TYPE

// ---- Abstractions/Components/MtsFeeding/Components/OscilatingConveyorFeeder/eTcoOscilatingConveyorStatus.TcDUT
{attribute 'qualified_only'}
{attribute 'strict'}
TYPE eTcoOscilatingConveyorStatus :
(
	None:=0,
	Feeding:=1,
	Oscilating:=2,
	ReadyToPick:=3,
	Error:=4

);
END_TYPE

// ---- Abstractions/Components/MtsFeeding/Components/OscilatingConveyorFeeder/TcoOscilatingConveyorFeederComponents.TcDUT
TYPE TcoOscilatingConveyorFeederComponents EXTENDS TcoCore.TcoStruct:
STRUCT


	

	
	
	{attribute wpf [Container(Layout.Stack,"Nasypnik")]}
	{attribute addProperty Name "<#Vstupny podavac prazdny#>"}
	iEntryFeederIsEmpty : TcoElements.TcoDi(THISSTRUCT);
	{attribute addProperty Name "<#Vstupny podavac preletovy senzor#>"}
	iFlowSensor : TcoElements.TcoDi(THISSTRUCT);
	
	{attribute addProperty Name "<#Vstupny podavac v chybe #>"}
	iEntryFeederError : TcoElements.TcoDi(THISSTRUCT);
	{attribute addProperty Name "<#Vyprazdnovaci box pritomny#>"}
	iThrowBoxPresent : TcoElements.TcoDi(THISSTRUCT);
	{attribute addProperty Name "<#Vstupny podavac Start #>"}
	qEntryFeederRun : TcoElements.TcoDo(THISSTRUCT);
	

	{attribute wpf [Container(Layout.Stack,"Dopravnik")]}
	{attribute addProperty Name "<#Oscilacny dopravnik je v chybe#>"}
	iOscConvError : TcoElements.TcoDi(THISSTRUCT);
	{attribute addProperty Name "<#Oscilacny dopravnik Start#>"}
	qOscConvRun : TcoElements.TcoDo(THISSTRUCT);
	{attribute addProperty Name "<#Oscilacny dopravnik reverz Start#>"}
	qOscConvRunReverse : TcoElements.TcoDo(THISSTRUCT);
	
	
	{attribute wpf [Container(Layout.Stack,"Valce")]}
	
	{attribute addProperty Name "<#Oscilacny cylinder  rad 1- vravo#>"}
	qOscCylinderRow1Right : TcoElements.TcoDo(THISSTRUCT);
	
	{attribute addProperty Name "<#Oscilacny cylinder rad 1 - vstrede#>"}
	qOscCylinderRow1Middle : TcoElements.TcoDo(THISSTRUCT);
	
	{attribute addProperty Name "<#Oscilacny cylinder rad 1 - vlavo#>"}
	qOscCylinderRow1Left : TcoElements.TcoDo(THISSTRUCT);
	
	{attribute addProperty Name "<#Oscilacny cylinder  rad 2- vravo#>"}
	qOscCylinderRow2Right : TcoElements.TcoDo(THISSTRUCT);
	
	{attribute addProperty Name "<#Oscilacny cylinder rad 2 - vstrede#>"}
	qOscCylinderRow2Middle : TcoElements.TcoDo(THISSTRUCT);
	
	{attribute addProperty Name "<#Oscilacny cylinder rad 2 - vlavo#>"}
	qOscCylinderRow2Left : TcoElements.TcoDo(THISSTRUCT);
	
	
	{attribute addProperty Name "<#Oscilacny cylinder  rad 3 - vravo#>"}
	qOscCylinderRow3Right : TcoElements.TcoDo(THISSTRUCT);
	
	{attribute addProperty Name "<#Oscilacny cylinder rad 3 - vstrede#>"}
	qOscCylinderRow3Middle : TcoElements.TcoDo(THISSTRUCT);
	
	{attribute addProperty Name "<#Oscilacny cylinder rad 3 - vlavo#>"}
	qOscCylinderRow3Left : TcoElements.TcoDo(THISSTRUCT);
	
	{attribute addProperty Name "<#Bocny matinel#>"}
	SideGuard : TcoPneumatics.TcoDoubleCylinder(THISSTRUCT);
	
	{attribute addProperty Name "<#Bocny matinel#>"}
	EntryFeederMantinel : TcoPneumatics.TcoCylinder(THISSTRUCT);


	{attribute wpf [Container(Layout.Stack,"Vseobecne")]}
	
	{attribute addProperty Name "(Q1) <#Signalizacia upozornenia R#>"}
	Q1_AttentionSignalisationR : TcoElements.TcoDo(THISSTRUCT);
	{attribute addProperty Name "(Q2) <#Signalizacia upozornenia G#>"}
	Q2_AttentionSignalisationG : TcoElements.TcoDo(THISSTRUCT);
	{attribute addProperty Name "(Q3) <#Signalizacia upozornenia B#>"}
	Q3_AttentionSignalisationB : TcoElements.TcoDo(THISSTRUCT);
	
	{attribute addProperty Name "<#Cognex Designer#>"}
	Designer : TcoCognexVision.TcoDesigner_v_2_x_x(THISSTRUCT);
END_STRUCT
END_TYPE

// ---- Abstractions/Components/MtsFeeding/Components/OscilatingConveyorFeeder/TcoOscilatingConveyorFeeder_Config_v_1_x_x.TcDUT
TYPE
    TcoOscilatingConveyorFeeder_Config_v_1_x_x EXTENDS TcoFeeding_Config_v_1_x_x :
    STRUCT
        {attribute addProperty Name "<#Ovladane kamerovym systemom#>"}
        ControledByVisonSystem : BOOL;

        {attribute addProperty Name "<#Oscilacny cylinder  rad 1- vravo#>"}
        EnableCylinderRow1Right : BOOL;

        {attribute addProperty Name "<#Oscilacny cylinder rad 1 - vstrede#>"}
        EnableCylinderRow1Middle : BOOL;

        {attribute addProperty Name "<#Oscilacny cylinder rad 1 - vlavo#>"}
        EnableCylinderRow1Left : BOOL;

        {attribute addProperty Name "<#Oscilacny cylinder  rad 2- vravo#>"}
        EnableCylinderRow2Right : BOOL;

        {attribute addProperty Name "<#Oscilacny cylinder rad 2 - vstrede#>"}
        EnableCylinderRow2Middle : BOOL;

        {attribute addProperty Name "<#Oscilacny cylinder rad 2 - vlavo#>"}
        EnableCylinderRow2Left : BOOL;

        {attribute addProperty Name "<#Oscilacny cylinder  rad 3- vravo#>"}
        EnableCylinderRow3Right : BOOL;

        {attribute addProperty Name "<#Oscilacny cylinder rad 3 - vstrede#>"}
        EnableCylinderRow3Middle : BOOL;

        {attribute addProperty Name "<#Oscilacny cylinder rad 3 - vlavo#>"}
        EnableCylinderRow3Left : BOOL;

        {attribute addProperty Name "<#Mantinel aktivny#>"}
        EnableSideGuard : BOOL;

        {attribute addProperty Name "<#Mantinel na dosipaci aktivny#>"}
        EnableEntryFeederMantinel : BOOL;

    //        {attribute addProperty Name "<#FillingTime#>"}
    //        FillingTime : TIME;

    //        {attribute addProperty Name "<#RunConv Time#>"}
    //        RunConvTime : TIME;

    //        {attribute addProperty Name "<#Oscilation Time #>"}
    //        OscilationTime : TIME;

    //        {attribute addProperty Name "<#Oscilation Type#>"}
    //        OscilationType : eTcoOscilatingConveyorOscilationModes;

    //        {attribute addProperty Name "<#Oscilation Frequency#>"}
    //        OscilationFreqency : TIME;

    //        {attribute addProperty Name "<#RunConvReverse Time#>"}
    //        RunConvRevTime : TIME;
    END_STRUCT
END_TYPE

// ---- Abstractions/Components/MtsFeeding/Components/OscilatingConveyorFeeder/TcoOscilatingConveyorFeeder_Control_v_1_x_x.TcDUT
TYPE TcoOscilatingConveyorFeeder_Control_v_1_x_x EXTENDS TcoCore.TcoStruct:
STRUCT

	
		
END_STRUCT
END_TYPE

// ---- Abstractions/Components/MtsFeeding/Components/OscilatingConveyorFeeder/TcoOscilatingConveyorFeeder_PcToPlc.TcDUT
TYPE TcoOscilatingConveyorFeeder_PcToPlc EXTENDS TcoCore.TcoStruct :
STRUCT
	EntryFeederRun : BOOL;
	OscConvRun : BOOL;
	OscConvRunReverse : BOOL;
	OscCylinderRow1Right : BOOL;
	OscCylinderRow1Middle : BOOL;
	OscCylinderRow1Left : BOOL;
	OscCylinderRow2Right : BOOL;
	OscCylinderRow2Middle : BOOL;
	OscCylinderRow2Left : BOOL;
	OscCylinderRow3Right : BOOL;
	OscCylinderRow3Middle : BOOL;
	OscCylinderRow3Left : BOOL;
	SideGuard : BOOL;
	EntryFeederMantinel : BOOL;
    Status : eTcoOscilatingConveyorStatus;
	StepDescription:STRING;
	ErrorDesription:STRING;

	
END_STRUCT
END_TYPE

// ---- Abstractions/Components/MtsFeeding/Components/OscilatingConveyorFeeder/TcoOscilatingConveyorFeeder_PlcToPc.TcDUT
TYPE
    TcoOscilatingConveyorFeeder_PlcToPc EXTENDS TcoCore.TcoStruct :
    STRUCT

        EntryFeederIsEmpty : BOOL;
        FlowSensor : BOOL;
        EntryFeederError : BOOL;
        ThrowBoxPresent : BOOL;
        OscConvError : BOOL;
        SideGuardAtHome : BOOL;
        SideGuardAtWork : BOOL;
        SafeCondition : BOOL;
        DoorOpen : BOOL;
        Mode : eCUMode;
        Config : TcoOscilatingConveyorFeeder_Config_v_1_x_x;
    END_STRUCT
END_TYPE

// ---- Abstractions/Components/MtsFeeding/Components/OscilatingConveyorFeeder/TcoOscilatingConveyorFeeder_Status_v_1_x_x.TcDUT
TYPE TcoOscilatingConveyorFeeder_Status_v_1_x_x EXTENDS TcoFeeding_Status_v_1_x_x:
STRUCT


		EntryBufferEmpty:BOOL;
		PcToPlcData:TcoOscilatingConveyorFeeder_PcToPlc;
		
END_STRUCT
END_TYPE

// ---- Abstractions/Components/Rework/eReworkResults.TcDUT
{attribute 'qualified_only'}
{attribute 'strict'}
TYPE eReworkResults :
(
	None:=0,
	Pass := 1,
	FailedEntityInProgress:=4,
	FailedEntityOk:=3,
	FailedEntityHasLessProgress:=2
	

);
END_TYPE

// ---- Abstractions/Components/Rework/ReworkData.TcDUT
TYPE ReworkData :
STRUCT
	{attribute addProperty Name "<#Entity Id#>"}
	EntityId: STRING;
	{attribute addProperty Name "<#ReworkId#>"}
	ReworkId: STRING;
	
	{attribute addProperty Name "<#Rework Instrukcia#>"}
	ReworkInstruction:STRING;
	{attribute addProperty Name "<#Rework Instrukcia najdena#>"}
	ReworkInstructionFound:BOOL;
	
END_STRUCT
END_TYPE

// ---- Abstractions/Components/TS/EqTransfer/eTcoEq2TransferConfiguration.TcDUT
{attribute 'qualified_only'}
{attribute 'strict'}
TYPE eTcoEq2TransferConfiguration :
(
	SingleInDoubleOut := 1,
	DoubleInSingleOut := 2,
	SingleInDoubleOutNoPrestopper := 3

);
END_TYPE

// ---- Abstractions/Components/TS/EqTransfer/eTcoEq2TransferHandlingMode.TcDUT
{attribute 'qualified_only'}
{attribute 'strict'}
TYPE eTcoEq2TransferHandlingMode :
(
	SendDirectWay := 1,
	SendSideWay := 2,
	RecieveDirectWay := 3,
	RecieveSideWay := 4

);
END_TYPE

// ---- Abstractions/Components/TS/EqTransfer/TcoEq2TransferComponents.TcDUT
TYPE
    TcoEq2TransferComponents EXTENDS TcoCore.TcoStruct :
    STRUCT
        {attribute addProperty Name "<#Pallete at prestopper - Main Transfer#>"}
        iPreStopperMainTransfer : TcoElements.TcoDi(THISSTRUCT);
        {attribute addProperty Name "<#Pallete at stopper - Main Transfer#>"}
        iStopperMainTransfer : TcoElements.TcoDi(THISSTRUCT);
        {attribute addProperty Name "<#Main Transfer is Empty#>"}
        iMainTransferIsEmpty : TcoElements.TcoDi(THISSTRUCT);
        {attribute addProperty Name "<#Output buffer full - Main Trasnfer#>"}
        iWipaMainTransfer : TcoElements.TcoDi(THISSTRUCT);
        {attribute addProperty Name "<#Prestopper - Main Transfer#>"}
        qPreStopperMainTransfer : TcoElements.TcoDo(THISSTRUCT);

        {attribute addProperty Name "<#Pallete at Prestopper Side transfer#>"}
        iPrestopperSideTransfer : TcoElements.TcoDi(THISSTRUCT);
        {attribute addProperty Name "<#Pallete at stopper Side transfer#>"}
        iStopperSideTransfer : TcoElements.TcoDi(THISSTRUCT);
        {attribute addProperty Name "<#Side Transfer is Empty#>"}
        iSideTransferIsEmpty : TcoElements.TcoDi(THISSTRUCT);
        {attribute addProperty Name "<#Out buffer full - Side Trasnfer#>"}
        iWipaSideTransfer : TcoElements.TcoDi(THISSTRUCT);
        {attribute addProperty Name "<#Prestopper Side transfer#>"}
        qPrestopperSideTransfer : TcoElements.TcoDo(THISSTRUCT);

		 {attribute addProperty Name "<#MotorInError#>"}
        iMotorError : TcoElements.TcoDi(THISSTRUCT);
        {attribute  addProperty Name "<#Motor#>"}
        qMotor : TcoElements.TcoDo(THISSTRUCT);
        {attribute addProperty Name "<#Transfer Position unit#>"}
        TransferUnit : TcoPneumatics.TcoCylinder(THISSTRUCT);

    END_STRUCT
END_TYPE

// ---- Abstractions/Components/TS/EqTransfer/TcoEq2Transfer_Config.TcDUT
TYPE
    TcoEq2Transfer_Config EXTENDS TcoCore.TcoStruct :
    STRUCT
     	InfoTime : TIME := T#5S;
        ErrorTime : TIME := T#0S;
        StabilisationTime : TIME := T#500MS;
		Mode:eTcoEq2TransferHandlingMode;
		Configuration:eTcoEq2TransferConfiguration;
    END_STRUCT
END_TYPE

// ---- Abstractions/Components/TS/EqTransfer/TcoEq2Transfer_Control.TcDUT
TYPE TcoEq2Transfer_Control EXTENDS TcoCore.TcoStruct:
STRUCT

	
		
END_STRUCT
END_TYPE

// ---- Abstractions/Components/TS/EqTransfer/TcoEq2Transfer_Status.TcDUT
TYPE TcoEq2Transfer_Status EXTENDS TcoCore.TcoStruct:
STRUCT


		ActionDescription:STRING;
		
END_STRUCT
END_TYPE

// ---- Abstractions/Components/TS/RotaryTrabsferWithLift/TcoLiftingRotaryTransferComponents.TcDUT
TYPE
    TcoLiftingRotaryTransferComponents EXTENDS TcoCore.TcoStruct :
    STRUCT

        {attribute addProperty Name "<#Paleta pred stanicou#>"}
        iPrestopper : TcoElements.TcoDi(THISSTRUCT);
        {attribute addProperty Name "<#Paleta v stanici#>"}
        iStopper : TcoElements.TcoDi(THISSTRUCT);
        {attribute addProperty Name "<#Transfer je prazdny#>"}
        iTransferIsEmpty : TcoElements.TcoDi(THISSTRUCT);

        {attribute addProperty Name "<#Vystup zo stanice plny#>"}
        iWipa : TcoElements.TcoDi(THISSTRUCT);
        {attribute addProperty Name "<#MotorInError#>"}
        iMotorError : TcoElements.TcoDi(THISSTRUCT);
        {attribute addProperty Name "<#Predzarazka#>"}
        qPrestopper : TcoElements.TcoDo(THISSTRUCT);
        {attribute  addProperty Name "<#Zarazka#>"}
        qStopper : TcoElements.TcoDo(THISSTRUCT);
        {attribute  addProperty Name "<#Motor#>"}
        qMotor : TcoElements.TcoDo(THISSTRUCT);
        {attribute addProperty Name "<Rotary unit#>"}
        RotaryUnit : TcoPneumatics.TcoCylinder(THISSTRUCT);
        {attribute addProperty Name "<#Vytah#>"}
        {attribute addProperty Retracted "<#Dole#>"}
        {attribute addProperty Extended "<#Hore#>"}
        {attribute addProperty Retracting "<#Pohyb dole#>"}
        {attribute addProperty Extending "<#Pohyb hore#>"}
        Lift : TcoPneumatics.TcoCylinder(THISSTRUCT);

    END_STRUCT
END_TYPE

// ---- Abstractions/Components/TS/RotaryTrabsferWithLift/TcoLiftingRotaryTransfer_Config.TcDUT
TYPE
    TcoLiftingRotaryTransfer_Config EXTENDS TcoCore.TcoStruct :
    STRUCT
     	InfoTime : TIME := T#5S;
        ErrorTime : TIME := T#0S;
        StabilisationTime : TIME := T#500MS;
		InvertLifting : BOOL;
	
		
    END_STRUCT
END_TYPE

// ---- Abstractions/Components/TS/RotaryTrabsferWithLift/TcoLiftingRotaryTransfer_Control.TcDUT
TYPE TcoLiftingRotaryTransfer_Control EXTENDS TcoCore.TcoStruct:
STRUCT

	
		
END_STRUCT
END_TYPE

// ---- Abstractions/Components/TS/RotaryTrabsferWithLift/TcoLiftingRotaryTransfer_Status.TcDUT
TYPE TcoLiftingRotaryTransfer_Status EXTENDS TcoCore.TcoStruct:
STRUCT


		ActionDescription:STRING;
		
END_STRUCT
END_TYPE

// ---- Abstractions/Components/TS/RotaryTransfer/TcoRotaryTransferComponents.TcDUT

TYPE
    TcoRotaryTransferComponents EXTENDS TcoCore.TcoStruct :
    STRUCT

        {attribute addProperty Name "<#Paleta pred stanicou#>"}
        iPrestopper : TcoElements.TcoDi(THISSTRUCT);
        {attribute addProperty Name "<#Paleta v stanici#>"}
        iStopper : TcoElements.TcoDi(THISSTRUCT);
        {attribute addProperty Name "<#Transfer je prazdny#>"}
        iTransferIsEmpty : TcoElements.TcoDi(THISSTRUCT);

        {attribute addProperty Name "<#Vystup zo stanice plny#>"}
        iWipa : TcoElements.TcoDi(THISSTRUCT);
        {attribute addProperty Name "<#MotorInError#>"}
        iMotorError : TcoElements.TcoDi(THISSTRUCT);
        {attribute addProperty Name "<#Predzarazka#>"}
        qPrestopper : TcoElements.TcoDo(THISSTRUCT);
        {attribute  addProperty Name "<#Zarazka#>"}
        qStopper : TcoElements.TcoDo(THISSTRUCT);
        {attribute  addProperty Name "<#Motor#>"}
        qMotor : TcoElements.TcoDo(THISSTRUCT);
        {attribute addProperty Name "<Rotary unit#>"}
        RotaryUnit : TcoPneumatics.TcoCylinder(THISSTRUCT);

    END_STRUCT
END_TYPE

// ---- Abstractions/Components/TS/RotaryTransfer/TcoRotaryTransfer_Config.TcDUT
TYPE
    TcoRotaryTransfer_Config EXTENDS TcoCore.TcoStruct :
    STRUCT
     	InfoTime : TIME := T#5S;
        ErrorTime : TIME := T#0S;
        StabilisationTime : TIME := T#500MS;
	
		
    END_STRUCT
END_TYPE

// ---- Abstractions/Components/TS/RotaryTransfer/TcoRotaryTransfer_Control.TcDUT
TYPE TcoRotaryTransfer_Control EXTENDS TcoCore.TcoStruct:
STRUCT

	
		
END_STRUCT
END_TYPE

// ---- Abstractions/Components/TS/RotaryTransfer/TcoRotaryTransfer_Status.TcDUT
TYPE TcoRotaryTransfer_Status EXTENDS TcoCore.TcoStruct:
STRUCT


		ActionDescription:STRING;
		
END_STRUCT
END_TYPE

// ---- Abstractions/Components/TS/WorkPosition/TcoTransferSystemComponents.TcDUT
TYPE TcoTransferSystemComponents EXTENDS TcoCore.TcoStruct:
STRUCT
	

	{attribute addProperty Name "<#Paleta pred stanicou#>"}
	iPrestopper  : TcoElements.TcoDi(THISSTRUCT);
	{attribute addProperty Name "<#Paleta v stanici#>"}
	iStopper     : TcoElements.TcoDi(THISSTRUCT);
	{attribute addProperty Name "<#Vystup zo stanice plny#>"}
	iWipa        : TcoElements.TcoDi(THISSTRUCT);
	{attribute addProperty Name "<#Predzarazka#>"}
	qPrestopper  : TcoElements.TcoDo(THISSTRUCT);
	{attribute  addProperty Name "<#Zarazka#>"}
	qStopper     : TcoElements.TcoDo(THISSTRUCT);
	{attribute addProperty Name "<#Pozicna jednotka#>"}
	{attribute addProperty Retracted "<#Dole#>"}
	{attribute addProperty Extended "<#Hore#>"}
	{attribute addProperty Retracting "<#Pohyb dole#>"}
	{attribute addProperty Extending "<#Pohyb hore#>"}
	PositionUnit : TcoPneumatics.TcoCylinder(THISSTRUCT);
	
	
	

	
	
END_STRUCT
END_TYPE

// ---- Abstractions/Components/TS/WorkPosition/TcoTransferSystem_Config.TcDUT
TYPE
    TcoTransferSystem_Config EXTENDS TcoCore.TcoStruct :
    STRUCT
     	InfoTime : TIME := T#5S;
        ErrorTime : TIME := T#0S;
        StabilisationTime : TIME := T#200MS;
		HasPositionUnit : BOOL :=TRUE;
		
    END_STRUCT
END_TYPE

// ---- Abstractions/Components/TS/WorkPosition/TcoTransferSystem_Control.TcDUT
TYPE TcoTransferSystem_Control EXTENDS TcoCore.TcoStruct:
STRUCT

	
		
END_STRUCT
END_TYPE

// ---- Abstractions/Components/TS/WorkPosition/TcoTransferSystem_Status.TcDUT
TYPE TcoTransferSystem_Status EXTENDS TcoCore.TcoStruct:
STRUCT


		ActionDescription:STRING;
		
END_STRUCT
END_TYPE

// ---- Abstractions/Components/WrappedComponent/WrappedComponentExample_Config.TcDUT
TYPE
    WrappedComponentExample_Config EXTENDS TcoCore.TcoStruct :
    STRUCT

        VacuumReachedStabilisation : TIME := T#100MS;
        VacuumPushTime : TIME := T#100MS;
    END_STRUCT
END_TYPE

// ---- Abstractions/Components/WrappedComponent/WrappedComponentExample_Control.TcDUT
TYPE WrappedComponentExample_Control EXTENDS TcoCore.TcoStruct:
STRUCT

		Setpoint:INT;
		
END_STRUCT
END_TYPE

// ---- Abstractions/Components/WrappedComponent/WrappedComponentExample_Status.TcDUT
TYPE WrappedComponentExample_Status EXTENDS TcoCore.TcoStruct:
STRUCT

		ProgressThrow:INT;
		ActionDescription:STRING;
END_STRUCT
END_TYPE

// ---- Abstractions/Components/WrappedComponent/WrappedComponentsExample.TcDUT
TYPE WrappedComponentsExample EXTENDS TcoCore.TcoStruct:
STRUCT
	
		{attribute addProperty Name "Vacuum Reached"}
		VacuumReached : TcoElements.TcoDi(THISSTRUCT);
		{attribute addProperty Name "Vacuum On"}
		VacuumOn : TcoElements.TcoDo(THISSTRUCT);
		{attribute addProperty Name "Vacuum Push"}
		VacuumPush : TcoElements.TcoDo(THISSTRUCT);
		
		{attribute addProperty Name "Gripper"}
		Gripper : TcoPneumatics.TcoCylinder(THISSTRUCT);
  
		{attribute addProperty Name "Manipulator"}
		Manipulator : TcoDrivesBeckhoff.TcoMultiAxis(THISSTRUCT);

		{attribute addProperty Name "Component Picked"}
		PresenceInGripper : TcoElements.TcoDi(THISSTRUCT);

	
	
END_STRUCT
END_TYPE

// ---- Abstractions/CUBase/CuBaseRecurringFail.TcDUT
TYPE CuBaseRecurringFail :
STRUCT
	Reached:BOOL;
	Result:TcoComprehensiveResult;
	Counter:UINT;
	
	
	
	
	
END_STRUCT
END_TYPE

// ---- Abstractions/CUBase/CuBaseRecurringFailures.TcDUT
TYPE CuBaseRecurringFailures EXTENDS TcoCore.TcoStruct : 
	STRUCT
   		AnyRecurringFails : CuBaseRecurringFail;
    	SameRecurringFails : CuBaseRecurringFail;
	END_STRUCT
END_TYPE

// ---- Abstractions/CUBase/CUBaseStatusInfo.TcDUT
TYPE
    CUBaseStatusInfo EXTENDS TcoCore.TcoStruct :
    STRUCT
     Mode                   : eCUMode;
     CurrentTaskDescription : STRING;
     CurrentUid             : INT;
     CurrentOperation       : STRING(255);
     CurrentCycleTime       : TIME;
	 AverageCycleTime       : TIME;
     CurrentIsInStepMode    : BOOL;
     CurrentCleanCycleTime  : TIME;
	 AverageCleanCycleTime  : TIME;
     State	                : eCUState;
     InSavingEnergy         : BOOL;
    END_STRUCT
END_TYPE

// ---- Abstractions/CUBase/CUBaseSettings.TcDUT
TYPE CUBaseSettings EXTENDS TcoCore.TcoStruct : STRUCT
    DeafultCycleTime : TIME;
    WarningCycleTime : TIME;
    ErrorCycleTime : TIME;
    SaveEnergyTime : TIME;
    AnyRecurringFailure : UINT;
    SameRecurringFailure : UINT;
END_STRUCT
END_TYPE

// ---- Abstractions/CUBase/Data/BasicCounterData.TcDUT
{attribute wpf [Container(Layout.Stack)]}
{attribute wpf [Group(Layout.Scroll)]}
{attribute addProperty Name "<#Entity header#>"}
TYPE BasicCounterData  EXTENDS TcoCore.TcoStruct :
STRUCT
	{attribute addProperty Name "<#OK#>"}
	Passed		: UDINT;
	{attribute addProperty Name "<#NOK#>"}
	Failed		: UDINT;
	{attribute addProperty Name "<#TOTAL#>"}
	Total		: UDINT;
	{attribute addProperty Name "<#ALL TIME OK#>"}
	LifeTimePassed	: UDINT;
	
	{attribute addProperty Name "<#ALL TIME NOK#>"}
	LifeTimeFailed	: UDINT;
	
	{attribute addProperty Name "<#ALL TIME #>"}
	LifeTime	: UDINT;
END_STRUCT
END_TYPE

// ---- Abstractions/CUBase/Data/CuHeader.TcDUT
TYPE CuHeader EXTENDS TcoCore.TcoStruct :
STRUCT
	{attribute addProperty Name "<#Next on Passed#>"}
	NextOnPassed : eStations;
	{attribute addProperty Name "<#Next on Failed#>"}
	NextOnFailed : eStations;
	{attribute clr [RenderIgnore("Control", "ShadowControl")]}
	{attribute addProperty Name "<#Cycle time#>"}
	CycleTime : TIME;
	{attribute clr [RenderIgnore("Control", "ShadowControl")]}
	{attribute addProperty Name "<#Clean loop time#>"}
	CleanLoopTime : TIME;
	{attribute clr [RenderIgnore("Control", "ShadowControl")]}
	{attribute addProperty Name "<#Operation started#>"}
	OperationsStarted : DT;
	{attribute clr [RenderIgnore("Control", "ShadowControl")]}
	{attribute addProperty Name "<#Operation ended#>"}
	OperationsEnded : DT;	
	{attribute clr [RenderIgnore("Control", "ShadowControl")]}
	{attribute addProperty Name "<#Operator#>"}
	Operator :STRING;	
END_STRUCT
END_TYPE

// ---- Abstractions/CUBase/Data/CUProcessDataBase.TcDUT
{attribute clr [Container(Layout.Stack)]}
{attribute clr [Group(Layout.Scroll)]}
TYPE CUProcessDataBase EXTENDS TcoCore.TcoStruct :
STRUCT
	{attribute wpf [Container(Layout.Stack)]}
	{attribute wpf [Group(Layout.GroupBox)]}
	Header : CuHeader := (Parent := THISSTRUCT);
END_STRUCT
END_TYPE

// ---- Abstractions/CUBase/Data/CUTechnologicalDataBase.TcDUT
{attribute clr [Container(Layout.Stack)]}
{attribute clr [Group(Layout.Scroll)]}
TYPE CUTechnologicalDataBase EXTENDS TcoCore.TcoStruct :
STRUCT
	{attribute wpf [Container(Layout.Stack,"General")]}
	{attribute wpf [Group(Layout.GroupBox)]}
	{attribute addProperty Name "<#Cycle time#> - <#Nominal#>"}
	IdealCycleTime   : TIME;
	
	
	{attribute addProperty Name "<#Cycle time#> - <#Warning#>"}
	WarningCycleTime : TIME;
    
	{attribute addProperty Name "<#Cycle time#> - <#Error#>"}
	ErrorCycleTime   : TIME;

	
	{attribute addProperty Name "<#Step time#> - <#Warning#>"}
	WarningStepAlarmTime : TIME;
    
	{attribute addProperty Name "<#Step time#> - <#Error#>"}
	ErrorStepAlarmTime   : TIME;
	
	{attribute addProperty Name "<#Energy saving mode - Inactivity time#>"}
	TimeToEntryEnergySavingMode : TIME;
	
	
	
	(*~
	<docu>
		<summary>
			The maximum allowed number of the any (arbitrary) recuring (consecutive)  failures.
		</summary>			
	</docu>	
	~*)
	{attribute addProperty Name "<#Max allowed number of any recurring failures (consecutive)#>"}
	AnyRecurringFailure   : UINT;
	
	

	(*~
	<docu>
		<summary>
			The maximum allowed number of the same (identical) recuring (consecutive) failures. 
		</summary>			
	</docu>	
	~*)
	{attribute addProperty Name "<#Max allowed number of same recurring failures (consecutive)#>"}
	SameRecurringFailure   : UINT;
	
	
END_STRUCT
END_TYPE

// ---- Abstractions/CUBase/Data/eCUState.TcDUT
{attribute 'qualified_only'}
{attribute 'strict'}
TYPE
    eCUState :
    (
        None       := 0,
        HasWarning := 10,
        HasError   := 20
    );
END_TYPE

// ---- Abstractions/CUBase/Data/eDataEntityInvokeType.TcDUT
{attribute 'qualified_only'}
{attribute 'strict'}
TYPE eDataEntityInvokeType : (
    InvokeAndWaitDone := 0,
    InvokeOnly	 := 10
);
END_TYPE

// ---- Abstractions/CUBase/Data/EntityHeader.TcDUT
{attribute wpf [Container(Layout.Stack)]}
{attribute wpf [Group(Layout.Scroll)]}
{attribute addProperty Name "<#Entity header#>"}
TYPE
    EntityHeader EXTENDS TcoCore.TcoStruct :
    STRUCT
        {attribute addProperty Name "<#Recipe#>"}
        {attribute clr [RenderIgnore("Control", "ShadowControl")]}
        Recipe : STRING(255);
        {attribute addProperty Name "<#Recipe created#>"}
        {attribute clr [RenderIgnore("Control", "ShadowControl")]}
        RecipeCreated : DT;
        {attribute addProperty Name "<#Recipe modified#>"}
        {attribute clr [RenderIgnore("Control", "ShadowControl")]}
        RecipeLastModified : DT;
        {attribute addProperty Name "<#Carrier#>"}
        {attribute clr [RenderIgnore("Control", "ShadowControl")]}
        Carrier : STRING;
        {attribute addProperty Name "<#Reset#>"}
        {attribute clr [RenderIgnore("Control", "ShadowControl")]}
        WasReset : BOOL;
        {attribute addProperty Name "<#Master#>"}
        {attribute clr [RenderIgnore("Control", "ShadowControl")]}
        IsMaster : BOOL;
        {attribute addProperty Name "<#Empty#>"}
        {attribute clr [RenderIgnore("Control", "ShadowControl")]}
        IsEmpty : BOOL;
        {attribute addProperty Name "<#Last station#>"}
        LastStation : eStations;
        {attribute addProperty Name "<#Next station#>"}
        NextStation : eStations;
        {attribute addProperty Name "<#Operations opened#>"}
        OpenOn : eStations;
        {attribute addProperty Name "<#Results#>"}
        Results : TcoInspectors.TcoComprehensiveResult;

        {attribute addProperty Name "<#Reworked#>"}
        {attribute clr [RenderIgnore("Control", "ShadowControl")]}
         WasReworked : BOOL;

        {attribute addProperty Name "<#Last Rework Name#>"}
        {attribute clr [RenderIgnore("Control", "ShadowControl")]}
         LastReworkName : STRING;

        {attribute addProperty Name "<#Rework Count#>"}
        {attribute clr [RenderIgnore("Control", "ShadowControl")]}
        ReworkCount : SINT;

    END_STRUCT
END_TYPE

// ---- Abstractions/Generic/LightTower/TcoLightTower_Config.TcDUT
TYPE
    TcoLightTower_Config :
    STRUCT
        MaxControledUnits : USINT := 12;
		HornEnabled:BOOL;
    END_STRUCT
END_TYPE

// ---- Abstractions/Generic/LightTower/TcoLightTower_Info.TcDUT
TYPE TcoLightTower_Info EXTENDS TcoControledZone_Info :
STRUCT

	
	
	{attribute addProperty Name "<#Group#> - <#Any station in warning#>"}
	AnyInWarning            : BOOL;
	
	{attribute addProperty Name "<#Group#> - <#Any station in error#>"}
	AnyInError          : BOOL;
	
	

END_STRUCT
END_TYPE

// ---- Abstractions/Generic/LightTower/TcoLightTower_Status.TcDUT
TYPE TcoLightTower_Status :
STRUCT
	ActionDescription : STRING(100);	
	State : TcoLightTower_Info;	
	
END_STRUCT
END_TYPE

// ---- Abstractions/Generic/NotificationPanel/NotificationPanelInfo.TcDUT
TYPE NotificationPanelInfo :
STRUCT
	{attribute addProperty Name "<#Control voltage#>"}
	ControlVoltage : BOOL;
	{attribute addProperty Name "<#Air pressure#>"}
	AirPressure : BOOL;
	{attribute addProperty Name "<#Autmatic mode allowed#>"}
	AutomatAllowed : BOOL;
	{attribute addProperty Name "<#Emergency stop#>"}
  	EmergencyStop : BOOL; 
	{attribute addProperty Name "<#Safety doors OK#>"}
  	SafetyDoorOk : BOOL;    
	{attribute addProperty Name "<#Doors closed#>"}
  	DoorClosed : BOOL;  
	{attribute addProperty Name "<#Doors locked#>"}
	DoorLocked : BOOL;
	{attribute addProperty Name "<#Light curtain#>"}
  	LightCurtain : BOOL;
	{attribute addProperty Name "<#Process data#>"}
  	ProcessDataOk : BOOL;
	{attribute addProperty Name "<#Technology data#>"}
  	TechnologyDataOk : BOOL;
END_STRUCT
END_TYPE

// ---- Abstractions/Generic/TagsPairing/eTagPairingAnswer.TcDUT
{attribute 'qualified_only'}
{attribute 'strict'}
TYPE
    eTagPairingAnswer :
    (
        TagFound := 0,
        TagFoundInactive := 10,
        TagFoundAssignedValueEmpty := 20,
        TagFoundUnknown := 30,
        TagNotFound := 40,
        TagAlreadyExist := 50,
        TagAddedSuccessfully := 60,
        TagAddedNotSuccessfuly := 70,
        EmptyCollection := 100
    );
END_TYPE

// ---- Abstractions/Generic/TagsPairing/eTagPairingMode.TcDUT
{attribute 'qualified_only'}
{attribute 'strict'}
TYPE
    eTagPairingMode :
    (
        GetTag := 1,
        RemoveTag := 2,
        AddTag := 3
    );
END_TYPE

// ---- Abstractions/Generic/TagsPairing/eTagPairingStatus.TcDUT
{attribute 'qualified_only'}
{attribute 'strict'}
TYPE
    eTagPairingStatus :
    (
        Unknown := 0,
        Active := 10,
        Inactive := 20
    );
END_TYPE

// ---- Abstractions/Generic/TagsPairing/TagsPairing.TcDUT
TYPE TagsPairing  EXTENDS TcoCore.TcoStruct :
STRUCT
	{attribute addProperty Name "<#Key UID#>"}
	Key : STRING;
	{attribute addProperty Name "<#Assigned Value#>"}
	AssignedValue : STRING;
	{attribute addProperty Name "<#Status#>"}
	Status : eTagPairingStatus;
	{attribute addProperty Name "<#Answer#>"}
	Answer : eTagPairingAnswer;
	
END_STRUCT
END_TYPE

// ---- Abstractions/Safety/ControlButtons/TcoControledZone_Info.TcDUT
TYPE TcoControledZone_Info :
STRUCT
	{attribute addProperty Name "<#All#> - <#In automatic#>"}
	AllInAuto            : BOOL;
	
	{attribute addProperty Name "<#All#> - <#Is grounding#>"}
	AllInGrounding       : BOOL;
	
	{attribute addProperty Name "<#All#> - <#In manual#>"}
	AllInManual          : BOOL;
	
	{attribute addProperty Name "<#All#> - <#Idle#>"}
	AllIdle          : BOOL;

	{attribute addProperty Name "<#All#> - <#Grounded#>"}
	AllGrounded          : BOOL;
	
	{attribute addProperty Name "<#All#> - <#In step mode#>"}
	AllInStepMode        : BOOL;
	
	{attribute addProperty Name "<#All#> - <#Recovered#>"}
	AllRecovered        : BOOL;
	
	{attribute addProperty Name "<#All#> - <#Suspended#>"}
	AllSuspended        : BOOL;
	
	{attribute addProperty Name "<#All#> - <#Holding process#>"}
	AllHolding           : BOOL;
	
	{attribute addProperty Name "<#All#> - <#In Inactive or Manual or Grounded#>"}
	AllInactiveOrManualOrGrounded  : BOOL;
	
	{attribute addProperty Name "<#Group#> - <#Any station in automatic mode#>"}
	AnyInAuto            : BOOL;
	
	{attribute addProperty Name "<#Group#> - <#Any station in manual mode#>"}
	AnyInManual          : BOOL;
	
	{attribute addProperty Name "<#Group#> - <#Any station in step mode#>"}
	AnyInStepMode        : BOOL;
	
	{attribute addProperty Name "<#Group#> - <#Any station is grounding#>"}
	AnyGrounding         : BOOL;
	
	{attribute addProperty Name "<#Group#> - <#Any station is holded#>"}
	AnyInHolding         : BOOL;
	
	{attribute addProperty Name "<#Control panel#> - <#All keys in automatic#>"}
	AllKeysAuto          : BOOL;
	
	{attribute addProperty Name "<#Control panel#> - <#All keys in normal#>"}
	AllKeysNormal        : BOOL;
	
	{attribute addProperty Name "<#Control panel#> - <#Any key in manual#>"}
	AnyKeyManual         : BOOL;
	
	{attribute addProperty Name "<#Control panel#> - <#Any key in step#>"}
	AnyKeyStep           : BOOL;
	
	{attribute addProperty Name "<#Control panel#> - <#Any key in service#>"}
	AnyKeyService        : BOOL;
	
	{attribute addProperty Name "<#Control panel#> - <#Any button#> - <#Recover#>"}
	AnyButtonRecover       : BOOL;
	
	{attribute addProperty Name "<#Control panel#> - <#Any button#> - <#Suspend#>"}
	AnyButtonSuspend        : BOOL;
	
	{attribute addProperty Name "<#Control panel#> - <#Any button#> - <#Ground#>"}
	AnyButtonGround      : BOOL;
	
	{attribute addProperty Name "<#Control panel#> - <#Any button#> - <#Auto#>"}
	AnyButtonAuto     : BOOL;
	
	{attribute addProperty Name "<#Deadman#> - <#Any present#>"}
	AnyDeadmanPresent    : BOOL;

END_STRUCT
END_TYPE

// ---- Abstractions/Safety/ControlledZone/TcoControlledZone_Config.TcDUT
TYPE
    TcoControlledZone_Config :
    STRUCT
        MaxControledUnits : USINT := 12;
        MaxControlButtons : USINT := 4;
        MaxKeyMode : USINT := 4;
        MaxKeyNormalService : USINT := 4;
        DoorsLocked : TIME := T#1S;
		AirPressureErrorTime : TIME :=T#5S;
    END_STRUCT
END_TYPE

// ---- Abstractions/Safety/ControlledZone/TcoControlledZone_Status.TcDUT
TYPE TcoControlledZone_Status :
STRUCT
	ActionDescription : STRING(100);	
	State : TcoControledZone_Info;	
	
END_STRUCT
END_TYPE

// ---- Abstractions/Safety/DoorCircuit/TcoDoorCircuit_Status.TcDUT
TYPE TcoDoorCircuit_Status :
STRUCT
	ActionDescription : STRING(100);	
END_STRUCT
END_TYPE

// ---- Abstractions/Safety/DoorCircuit/TcoDoorCircuit_Config.TcDUT
TYPE
    TcoDoorCircuit_Config :
    STRUCT
        InfoTime : TIME := T#2S;
        ErrorTime : TIME := T#0S;
		MaxDoors : USINT:=12;
		MaxLocalDoorsVoltage : USINT:=4;
		MaxLocalVoltage: USINT:=4;
		MaxGlobalVoltage: USINT:=4;
	
    END_STRUCT
END_TYPE

// ---- Abstractions/Safety/KeyMode/TcoKeyMode_Config.TcDUT
TYPE
    TcoKeyMode_Config :
    STRUCT
        SwitKeyStanilisiation : TIME := T#500mS;

	
    END_STRUCT
END_TYPE

// ---- Abstractions/Safety/KeyMode/TcoKeyMode_Status.TcDUT
TYPE TcoKeyMode_Status :
STRUCT
	ActionDescription : STRING(100);	

END_STRUCT
END_TYPE

// ---- Abstractions/TcoCore/CycleTimeAnalitics.TcDUT
TYPE CycleTimeAnalitics :
STRUCT

	{attribute addProperty Name "<#Average cycle time#>"}
	Average:TIME;
	
	{attribute addProperty Name "<#Average clean cycle time#>"}
	AverageCleanCycle:TIME;
	
	{attribute addProperty Name "<#Average cycle time filter constant#>"}
	FilterConstant:UINT:=10;	
	

	
END_STRUCT
END_TYPE

// ---- DUTs/IO_Specific/Aventics/AES_D_BC_ECAT_Gen2_32bytes_Data_Inputs.TcDUT
{attribute 'GeneratedUsingTerminal: AES-D-BC-ECAT Gen2-0001'}
{attribute addProperty BoxType "AES-D-BC-ECAT Gen2-0001"}
{attribute addProperty Id "digital_Data_IAT %I*ARRAY[0..31] OF ARRAY[0..7] OF BOOL"}
{attribute addProperty CRC "1374483313"}
{attribute addProperty Size "32"}
TYPE AES_D_BC_ECAT_Gen2_32bytes_Data_Inputs EXTENDS TcoIo.InputBase_8311D824 :
STRUCT
	{attribute addProperty Name "digital_Data_I"}
	digital_Data_I AT %I* : ARRAY[0..31] OF ARRAY[0..7] OF BOOL;
END_STRUCT
END_TYPE

// ---- DUTs/IO_Specific/Aventics/AES_D_BC_ECAT_Gen2_32bytes_Data_Outputs.TcDUT
{attribute 'GeneratedUsingTerminal: AES-D-BC-ECAT Gen2-0001'}
{attribute addProperty BoxType "AES-D-BC-ECAT Gen2-0001"}
{attribute addProperty Id "digital_Data_OAT %Q*ARRAY[0..31] OF ARRAY[0..7] OF BOOL"}
{attribute addProperty CRC "2024821696"}
{attribute addProperty Size "32"}
TYPE AES_D_BC_ECAT_Gen2_32bytes_Data_Outputs EXTENDS TcoIo.OutputBase_10CEE7DE :
STRUCT
	{attribute addProperty Name "digital_Data_O"}
	digital_Data_O AT %Q* : ARRAY[0..31] OF ARRAY[0..7] OF BOOL;
END_STRUCT
END_TYPE

// ---- DUTs/IO_Specific/Aventics/AES_D_BC_ECAT_Gen2_4bytes_Data_Inputs.TcDUT
{attribute 'GeneratedUsingTerminal: AES-D-BC-ECAT Gen2-0001'}
{attribute addProperty BoxType "AES-D-BC-ECAT Gen2-0001"}
{attribute addProperty Id "digital_Data_IAT %I*ARRAY[0..3] OF ARRAY[0..7] OF BOOL"}
{attribute addProperty CRC "753485497"}
{attribute addProperty Size "4"}
TYPE AES_D_BC_ECAT_Gen2_4bytes_Data_Inputs EXTENDS TcoIo.InputBase_8311D824 :
STRUCT
	{attribute addProperty Name "digital_Data_I"}
	digital_Data_I AT %I* : ARRAY[0..3] OF ARRAY[0..7] OF BOOL;
END_STRUCT
END_TYPE

// ---- DUTs/IO_Specific/Aventics/AES_D_BC_ECAT_Gen2_4bytes_Data_Outputs.TcDUT
{attribute 'GeneratedUsingTerminal: AES-D-BC-ECAT Gen2-0001'}
{attribute addProperty BoxType "AES-D-BC-ECAT Gen2-0001"}
{attribute addProperty Id "digital_Data_OAT %Q*ARRAY[0..3] OF ARRAY[0..7] OF BOOL"}
{attribute addProperty CRC "2104334051"}
{attribute addProperty Size "4"}
TYPE AES_D_BC_ECAT_Gen2_4bytes_Data_Outputs EXTENDS TcoIo.OutputBase_10CEE7DE :
STRUCT
	{attribute addProperty Name "digital_Data_O"}
	digital_Data_O AT %Q* : ARRAY[0..3] OF ARRAY[0..7] OF BOOL;
END_STRUCT
END_TYPE

// ---- Technology/CU00x/Components/CU00xExamplesOfComponents.TcDUT
{attribute wpf [Container(Layout.Stack)]}	
{attribute wpf [Group(Layout.Scroll)]}
TYPE CU00xExamplesOfComponents EXTENDS TcoCore.TcoStruct:
STRUCT
		{attribute wpf [Container(Layout.Stack,"PNEU")]}	
		{attribute addProperty Name "(A1)HORIZONTAL AXIS"}
      	horizontalCylinder : TcoPneumatics.TcoCylinder(THISSTRUCT); 
		{attribute addProperty Name "(A2)VERTICAL AXIS"}
      	verticalCylinder : TcoPneumatics.TcoCylinder(THISSTRUCT); 
		
		{attribute addProperty Name "(A3)DOUBLE "}
      	doubleCylinder : TcoPneumatics.TcoDoubleCylinder(THISSTRUCT); 
		
		{attribute wpf [Container(Layout.Stack,"INPUTS")]}	
		{attribute addProperty Name "PRESENCE ON INSPECTION"}
     	PresenceOnInspection : TcoElements.TcoDi(THISSTRUCT);
		
		{attribute addProperty Name "PRESENCE AT ENTRY CONVEYOR"}
     	PresenceComponentAtEntr: TcoElements.TcoDi(THISSTRUCT);
		
		{attribute addProperty Name "COLISION SENSOR"}
     	ColisonSensorComponent: TcoElements.TcoDi(THISSTRUCT);

		{attribute addProperty Name "CONVEYOR AT ENTRY IS EMPTY"}
     	ConvAtEntryIsEmpty : TcoElements.TcoDi(THISSTRUCT);
		
		{attribute addProperty Name "INSPECTION NOK"}
     	InspectionIsNok : TcoElements.TcoDi(THISSTRUCT);
		

		{attribute wpf [Container(Layout.Stack,"OUTPUTS")]}		
		{attribute addProperty Name "LIGHT ON"}
     	LightOn : TcoElements.TcoDi(THISSTRUCT); 
		
		{attribute addProperty Name "LIGHT OFF"}
     	LightOff : TcoElements.TcoDi(THISSTRUCT);
		{attribute wpf [Container(Layout.Stack,"ANALOGS")]}	
		{attribute addProperty Name "VERIFY SETPOINT"}
     	VerifySetpoint : TcoElements.TcoAi(THISSTRUCT);
		{attribute addProperty Name "SETPOINT"}
     	Setpoint : TcoElements.TcoAo(THISSTRUCT);   
		
		{attribute addProperty Name "SampleDataToRender"}
     	ArrayToRender : SampleArrayToRender;   

END_STRUCT
END_TYPE

// ---- Technology/CU00x/Data/CU00xTechnologicalData.TcDUT
TYPE
    CU00xTechnologicalData EXTENDS CUTechnologicalDataBase : 
    STRUCT		
		{attribute wpf [Container(Layout.Stack,"Station specific data")]}
		{attribute wpf [Group(Layout.GroupBox)]}
		{attribute addProperty Name "Axis Home position"}
        ServoHomePosition : LREAL;
		{attribute addProperty Name "Axis Work position"}
		ServoWorkPosition : LREAL;
    END_STRUCT
END_TYPE

// ---- Technology/Data/ProcessData.TcDUT
{attribute clr [Container(Layout.Tabs)]}
TYPE
    ProcessData EXTENDS TcoEntityBase :
    STRUCT

        {attribute addProperty Name "<#Entity header#>"}
        EntityHeader : EntityHeader     := (Parent := THISSTRUCT);
		{attribute addProperty Name "<#CU00x#>"}
		{attribute clr [Container(Layout.Stack)]}
        CU00x : CU00xProcessData := (Parent := THISSTRUCT);
    END_STRUCT
END_TYPE

// ---- Technology/CU00x/Components/CU00xComponents.TcDUT
{attribute wpf [Container(Layout.Tabs)]}
TYPE
    CU00xComponents EXTENDS CUComponentsBase :
    STRUCT
		{attribute wpf [Container(Layout.Stack)]}
		{attribute wpf [Group(Layout.Scroll)]}
		{attribute addProperty Name "Supplu TTI QL"}
     	Supply : TcoAimTtiPowerSupply.TcoQl355P_v_1_x_x (THISSTRUCT);
		{attribute wpf [Container(Layout.Stack)]}
		PairTagTask: PairTagTask(THISSTRUCT);
		{attribute wpf [Container(Layout.Stack)]}
		{attribute addProperty Name "<#ReworkInstruction#>"}
		ReworkInstructionTask : ReworkInstructionTask(THISSTRUCT);
		{attribute wpf [Container(Layout.Stack,"DRIVES AND MANIPULATORS")]}	
		{attribute wpf [Group(Layout.Scroll)]}
		{attribute addProperty Name "MultiAxis"}
     	MultiAxis : TcoDrivesBeckhoff.TcoMultiAxis(THISSTRUCT);
		{attribute addProperty Name "Single Axis"}
     	SingleAxis : TcoDrivesBeckhoff.TcoSingleAxis(THISSTRUCT);
		{attribute addProperty Name "Simple drive"}
     	SimpleDrive : TcoDrivesBeckhoff.TcoDriveSimple(THISSTRUCT);
		
		{attribute wpf [Container(Layout.Stack,"VISION")]}	
		{attribute wpf [Group(Layout.Scroll)]}
		{attribute addProperty Name "Dataman"}
     	Dmc : TcoCognexVision.TcoDataman_v_5_x_x(THISSTRUCT);
		{attribute addProperty Name "Insight"}
     	Cam : TcoCognexVision.TcoInsight_v_5_x_x(THISSTRUCT);

	
		{attribute wpf [Container(Layout.Stack,"ROBOTICS")]}	
		{attribute wpf [Group(Layout.Scroll)]}
		{attribute addProperty Name "Abb IRC 5"}
     	AbbIrc5 : TcoAbbRobotics.TcoIrc5_v_1_x_x(THISSTRUCT);
		{attribute addProperty Name "Abb Omnicore"}
     	AbbOmnicore : TcoAbbRobotics.TcoOmnicore_v_1_x_x(THISSTRUCT);
		
		{attribute addProperty Name "Mitshubishi Cr series"}
     	MitshubishiCr: TcoMitsubishiRobotics.TcoCr800_v_1_x_x(THISSTRUCT);
		{attribute addProperty Name "UR CB series"}
     	UrCb3:  TcoUrRobotics.TcoUrCb3_v_3_x_x(THISSTRUCT);
		{attribute addProperty Name "Ur E series"}
     	UrEseries: TcoUrRobotics.TcoUrEseries_v_5_x_x(THISSTRUCT);
		
		{attribute addProperty Name "Kuka Krc4"}
     	KukaKrc4: TcoKukaRobotics.TcoKrc4_v_5_x_x(THISSTRUCT);
		
		{attribute wpf [Container(Layout.Stack,"TIXONS")]}	
		{attribute wpf [Group(Layout.Scroll)]}
		{attribute addProperty Name "Tixon Vibro"}
     	TixonVibro : TcoTixonFeeding.TcoTixonVibro_v_1_x_x(THISSTRUCT);
		{attribute addProperty Name "Tixon Step"}
     	TixonStep : TcoTixonFeeding.TcoTixonStep_v_1_x_x(THISSTRUCT);
		
		{attribute addProperty Name "Tixon Pick Vibro"}
     	TixonPickVibro : TcoTixonFeeding.TcoTixonPickVibro_v_1_x_x(THISSTRUCT);
		{attribute addProperty Name "Tixon Pick Step"}
     	TixonPickStep : TcoTixonFeeding.TcoTixonPickStep_v_1_x_x(THISSTRUCT);
			
		{attribute wpf [Container(Layout.Stack,"MtsFeeding")]}	
		{attribute wpf [Group(Layout.Scroll)]}
		PlsPaletizator:TcoPlsPaletizator(THISSTRUCT);	
		{attribute clr [RenderIgnore()]}
		PlsPaletizatorComponents:TcoPlsPaletizator_Components := (Parent := THISSTRUCT);  
		
		{attribute wpf [Group(Layout.Scroll)]}
		PlrPaletizator:TcoPlrPaletizator(THISSTRUCT);	
		{attribute clr [RenderIgnore()]}
		PlrPaletizatorComponents:TcoPlrPaletizator_Components := (Parent := THISSTRUCT);  
		
		{attribute wpf [Group(Layout.Scroll)]}
		PlbPaletizator:TcoPlbPaletizator(THISSTRUCT);	
		{attribute clr [RenderIgnore()]}
		PlbPaletizatorComponents:TcoPlbPaletizator_Components := (Parent := THISSTRUCT);  
		
		
		{attribute wpf [Container(Layout.Stack)]}
        {attribute wpf [Group(Layout.Scroll)]}
        OscilatingFeeder : TcoOscilatingConveyorFeeder(THISSTRUCT);
        {attribute clr [RenderIgnore()]}
        OscilatingFeederComponents : TcoOscilatingConveyorFeederComponents := (Parent := THISSTRUCT);

		
		{attribute wpf [Container(Layout.Stack,"Wrapped component example")]}	
		{attribute wpf [Group(Layout.Scroll)]}
		PickAndPlace:WrappedComponentExample(THISSTRUCT);
		{attribute wpf [Container(Layout.Stack,"Wrapped component struct")]}	
		PickAndPlaceCompoennts:WrappedComponentsExample := (Parent := THISSTRUCT);  

		{attribute addProperty Name "GROUP 1"}
		Group1 : CU00xExamplesOfComponents := (Parent := THISSTRUCT);  
		{attribute addProperty Name "GROUP 2"}
		Group2 : CU00xExamplesOfComponents := (Parent := THISSTRUCT); 
 
    END_STRUCT
END_TYPE

// ---- Technology/CU00x/Data/CU00xProcessData.TcDUT
TYPE
    CU00xProcessData EXTENDS CUProcessDataBase :
    STRUCT
		{attribute wpf [Container(Layout.Stack)]}
		{attribute addProperty Name "Bolt present inspection"}
        BoltPresenceInspector : TcoInspectors.TcoDigitalInspector(THISSTRUCT);
		{attribute addProperty Name "Bolt Dimension inspection"}
		BoltDimensionPresenceInspector : TcoInspectors.TcoAnalogueInspector(THISSTRUCT);
		{attribute addProperty Name "Bolt code inspection"}
		BoltDatacodePresenceInspector : TcoInspectors.TcoDataInspector(THISSTRUCT);

		{attribute addProperty Name "Dimension inspection 1"}
        Dim_Inspector_1 : TcoInspectors.TcoAnalogueInspector(THISSTRUCT);
		{attribute addProperty Name "Dimension inspection 2"}
        Dim_Inspector_2 : TcoInspectors.TcoAnalogueInspector(THISSTRUCT);
		{attribute addProperty Name "Dimension inspection 3"}
		Dim_Inspector_3 : TcoInspectors.TcoAnalogueInspector(THISSTRUCT);
		{attribute addProperty Name "Dimension inspection 4"}
        Dim_Inspector_4 : TcoInspectors.TcoAnalogueInspector(THISSTRUCT);
		{attribute addProperty Name "Dimension inspection 5"}
        Dim_Inspector_5 : TcoInspectors.TcoAnalogueInspector(THISSTRUCT);
		{attribute addProperty Name "Dimension inspection 6"}
        Dim_Inspector_6 : TcoInspectors.TcoAnalogueInspector(THISSTRUCT);
		{attribute addProperty Name "Dimension inspection 7"}
        Dim_Inspector_7 : TcoInspectors.TcoAnalogueInspector(THISSTRUCT);
		{attribute addProperty Name "Dimension inspection 8"}
        Dim_Inspector_8 : TcoInspectors.TcoAnalogueInspector(THISSTRUCT);
		{attribute addProperty Name "Dimension inspection 9"}
        Dim_Inspector_9 : TcoInspectors.TcoAnalogueInspector(THISSTRUCT);
		{attribute addProperty Name "Dimension inspection 10"}
        Dim_Inspector_10 : TcoInspectors.TcoAnalogueInspector(THISSTRUCT);
		
		{attribute addProperty Name "Dimension inspection 11"}
        Dim_Inspector_11 : TcoInspectors.TcoAnalogueInspector(THISSTRUCT);
		{attribute addProperty Name "Dimension inspection 12"}
        Dim_Inspector_12 : TcoInspectors.TcoAnalogueInspector(THISSTRUCT);
		{attribute addProperty Name "Dimension inspection 13"}
		Dim_Inspector_13 : TcoInspectors.TcoAnalogueInspector(THISSTRUCT);
		{attribute addProperty Name "Dimension inspection 14"}
        Dim_Inspector_14 : TcoInspectors.TcoAnalogueInspector(THISSTRUCT);
		{attribute addProperty Name "Dimension inspection 15"}
        Dim_Inspector_15 : TcoInspectors.TcoAnalogueInspector(THISSTRUCT);
		{attribute addProperty Name "Dimension inspection 16"}
        Dim_Inspector_16 : TcoInspectors.TcoAnalogueInspector(THISSTRUCT);
		{attribute addProperty Name "Dimension inspection 17"}
        Dim_Inspector_17 : TcoInspectors.TcoAnalogueInspector(THISSTRUCT);
		{attribute addProperty Name "Dimension inspection 18"}
        Dim_Inspector_18 : TcoInspectors.TcoAnalogueInspector(THISSTRUCT);
		{attribute addProperty Name "Dimension inspection 19"}
        Dim_Inspector_19 : TcoInspectors.TcoAnalogueInspector(THISSTRUCT);
		{attribute addProperty Name "Dimension inspection 20"}
        Dim_Inspector_20 : TcoInspectors.TcoAnalogueInspector(THISSTRUCT);
    END_STRUCT
END_TYPE

// ---- Technology/Data/TcoEntityBase.TcDUT
TYPE TcoEntityBase EXTENDS TcoData.TcoEntity :
STRUCT
	{attribute clr [RenderIgnore("Control", "ShadowControl")]}
	{attribute addProperty Name "<#Created#>"}
	_Created : DT;
	{attribute clr [RenderIgnore("Control", "ShadowControl")]}
	{attribute addProperty Name "<#Modified#>"}
	_Modified : DT;
END_STRUCT
END_TYPE

// ---- Technology/Data/TechnologyData.TcDUT
{attribute clr [Container(Layout.Tabs)]}
TYPE
    TechnologyData EXTENDS TcoEntityBase :
    STRUCT

        CU00x : CU00xTechnologicalData := (Parent := THISSTRUCT);
    END_STRUCT
END_TYPE

// ---- Technology/TechnologyComponents.TcDUT
{attribute wpf [Container(Layout.Tabs)]}
TYPE
    TechnologyComponents EXTENDS TcoCore.TcoStruct :
    STRUCT
      	{attribute wpf [Container(Layout.Stack,"PRESURE")]}
        {attribute addProperty Name "<#Presure OK#>"}
        AirPresureOk : TcoElements.TcoDi(THISSTRUCT);  
	
		{attribute wpf [Container(Layout.Stack,"ESTOPS")]}
        {attribute addProperty Name "<#Emergency Stop#>"}
        EmergencyStop : TcoEmergencyStop(THISSTRUCT);

		{attribute wpf [Container(Layout.Stack,"CONTROL VOLTAGE")]}
        {attribute addProperty Name "<#Global control voltage#>"}
        GlobalControlVoltage : TcoControlVoltage(THISSTRUCT);
		

        {attribute addProperty Name "<#Local control voltage#>"}
        LocalControlVoltage : TcoControlVoltage(THISSTRUCT);
		

        {attribute addProperty Name "<#Local door voltage#>"}
        LocalDoorVoltage : TcoControlVoltage(THISSTRUCT);
		
		
		{attribute wpf [Container(Layout.Stack,"CONTROLS")]}
        {attribute addProperty Name "<#Control Buttons#>"}
        ControlButtons : TcoControlButtons(THISSTRUCT);
		
        {attribute addProperty Name "<#Mode key#>"}
        ModeKey : TcoKeyMode(THISSTRUCT);
		
		{attribute addProperty Name "<#Normal/Service key#>"}
        NormalServiceKey : TcoKeyNormalService(THISSTRUCT);
		
		{attribute wpf [Container(Layout.Stack,"DOORS")]}
		{attribute addProperty Name "<#Standard door#>"}
        StandardDoor : TcoStandardDoor(THISSTRUCT);

		{attribute addProperty Name "<#Basic door#>"}
        BasicDoor : TcoBasicDoor(THISSTRUCT);

		
		{attribute wpf [Container(Layout.Stack,"DOORCIRUITS AND ZONES")]}
		{attribute addProperty Name "<#Door circuit#>"}
        DoorCicuit : TcoDoorCircuit(THISSTRUCT);

		
		{attribute addProperty Name "<#Zone#>"}
        Zone : TcoControlledZone(THISSTRUCT);



    END_STRUCT
END_TYPE

// ---- DUTs/IO/PDOs/Channel_830843C1.TcDUT
{attribute 'GeneratedUsingTerminal: EL1809-0000-0018'}
{attribute addProperty BoxType "EL1809-0000-0018"}
{attribute addProperty Id "InputAT %I*BOOL1"}
{attribute addProperty CRC "2198356929"}
{attribute addProperty Size "1"}
TYPE Channel_830843C1 EXTENDS TcoIo.InputBase_8311D824 :
STRUCT
	{attribute addProperty Name "Input"}
	Input AT %I* : BOOL;
END_STRUCT
END_TYPE

// ---- DUTs/IO/PDOs/Channel_42CA91F7.TcDUT
{attribute 'GeneratedUsingTerminal: EL2809-0000-0018'}
{attribute addProperty BoxType "EL2809-0000-0018"}
{attribute addProperty Id "OutputAT %Q*BOOL1"}
{attribute addProperty CRC "1120571895"}
{attribute addProperty Size "1"}
TYPE Channel_42CA91F7 EXTENDS TcoIo.OutputBase_10CEE7DE :
STRUCT
	{attribute addProperty Name "Output"}
	Output AT %Q* : BOOL;
END_STRUCT
END_TYPE

// ---- DUTs/IO/Boxes/EK1200_013D0B49.TcDUT
{attribute 'GeneratedUsingTerminal: EK1200-1388-0000'}
{attribute addProperty VendorId "#x00000002"}
{attribute addProperty BoxType "EK1200-1388-0000"}
{attribute addProperty Description "EK1200-5000 EtherCAT Power supply (2A E-Bus)"}
{attribute addProperty Physics "YK"}
{attribute addProperty Id "EK1200"}
{attribute addProperty CRC "20777801"}
{attribute addProperty Size "0"}
TYPE EK1200_013D0B49 EXTENDS TcoIo.EtcSlaveBoxBase_77A0E4A7 :
STRUCT
END_STRUCT
END_TYPE

// ---- DUTs/IO/Boxes/EK1122_1FC0878B.TcDUT
{attribute 'GeneratedUsingTerminal: EK1122-0000-0018'}
{attribute addProperty VendorId "#x00000002"}
{attribute addProperty BoxType "EK1122-0000-0018"}
{attribute addProperty Description "EK1122 2 port EtherCAT junction"}
{attribute addProperty Physics "KYKY"}
{attribute addProperty Id "InfoDataAT %I*InfoData_6F19DB2B2"}
{attribute addProperty CRC "532711307"}
{attribute addProperty Size "2"}
TYPE EK1122_1FC0878B EXTENDS TcoIo.EtcSlaveTerminalBase_947E5A46 :
STRUCT
	{attribute addProperty Name "InfoData"}
	InfoData : TcoIo.InfoData_6F19DB2B;
END_STRUCT
END_TYPE

// ---- DUTs/IO/Boxes/EL1809_32157CFD.TcDUT
{attribute 'GeneratedUsingTerminal: EL1809-0000-0018'}
{attribute addProperty VendorId "#x00000002"}
{attribute addProperty BoxType "EL1809-0000-0018"}
{attribute addProperty Description "EL1809 16Ch. Dig. Input 24V, 3ms"}
{attribute addProperty Physics "KK"}
{attribute addProperty Id "Channel_1AT %I*Channel_830843C11Channel_2AT %I*Channel_830843C11Channel_3AT %I*Channel_830843C11Channel_4AT %I*Channel_830843C11Channel_5AT %I*Channel_830843C11Channel_6AT %I*Channel_830843C11Channel_7AT %I*Channel_830843C11Channel_8AT %I*Channel_830843C11Channel_9AT %I*Channel_830843C11Channel_10AT %I*Channel_830843C11Channel_11AT %I*Channel_830843C11Channel_12AT %I*Channel_830843C11Channel_13AT %I*Channel_830843C11Channel_14AT %I*Channel_830843C11Channel_15AT %I*Channel_830843C11Channel_16AT %I*Channel_830843C11WcStateAT %I*WcState_9091E0EB2InfoDataAT %I*InfoData_6F19DB2B2"}
{attribute addProperty CRC "840269053"}
{attribute addProperty Size "20"}
TYPE EL1809_32157CFD EXTENDS TcoIo.EtcSlaveTerminalBase_947E5A46 :
STRUCT
	{attribute addProperty Name "Channel_1"}
	Channel_1 : Channel_830843C1;
	{attribute addProperty Name "Channel_2"}
	Channel_2 : Channel_830843C1;
	{attribute addProperty Name "Channel_3"}
	Channel_3 : Channel_830843C1;
	{attribute addProperty Name "Channel_4"}
	Channel_4 : Channel_830843C1;
	{attribute addProperty Name "Channel_5"}
	Channel_5 : Channel_830843C1;
	{attribute addProperty Name "Channel_6"}
	Channel_6 : Channel_830843C1;
	{attribute addProperty Name "Channel_7"}
	Channel_7 : Channel_830843C1;
	{attribute addProperty Name "Channel_8"}
	Channel_8 : Channel_830843C1;
	{attribute addProperty Name "Channel_9"}
	Channel_9 : Channel_830843C1;
	{attribute addProperty Name "Channel_10"}
	Channel_10 : Channel_830843C1;
	{attribute addProperty Name "Channel_11"}
	Channel_11 : Channel_830843C1;
	{attribute addProperty Name "Channel_12"}
	Channel_12 : Channel_830843C1;
	{attribute addProperty Name "Channel_13"}
	Channel_13 : Channel_830843C1;
	{attribute addProperty Name "Channel_14"}
	Channel_14 : Channel_830843C1;
	{attribute addProperty Name "Channel_15"}
	Channel_15 : Channel_830843C1;
	{attribute addProperty Name "Channel_16"}
	Channel_16 : Channel_830843C1;
	{attribute addProperty Name "WcState"}
	WcState : TcoIo.WcState_9091E0EB;
	{attribute addProperty Name "InfoData"}
	InfoData : TcoIo.InfoData_6F19DB2B;
END_STRUCT
END_TYPE

// ---- DUTs/IO/Boxes/EL2809_2B6483BD.TcDUT
{attribute 'GeneratedUsingTerminal: EL2809-0000-0018'}
{attribute addProperty VendorId "#x00000002"}
{attribute addProperty BoxType "EL2809-0000-0018"}
{attribute addProperty Description "EL2809 16Ch. Dig. Output 24V, 0.5A"}
{attribute addProperty Physics "KK"}
{attribute addProperty Id "Channel_1AT %Q*Channel_42CA91F71Channel_2AT %Q*Channel_42CA91F71Channel_3AT %Q*Channel_42CA91F71Channel_4AT %Q*Channel_42CA91F71Channel_5AT %Q*Channel_42CA91F71Channel_6AT %Q*Channel_42CA91F71Channel_7AT %Q*Channel_42CA91F71Channel_8AT %Q*Channel_42CA91F71Channel_9AT %Q*Channel_42CA91F71Channel_10AT %Q*Channel_42CA91F71Channel_11AT %Q*Channel_42CA91F71Channel_12AT %Q*Channel_42CA91F71Channel_13AT %Q*Channel_42CA91F71Channel_14AT %Q*Channel_42CA91F71Channel_15AT %Q*Channel_42CA91F71Channel_16AT %Q*Channel_42CA91F71WcStateAT %I*WcState_0B2B16F91InfoDataAT %I*InfoData_6F19DB2B2"}
{attribute addProperty CRC "728007613"}
{attribute addProperty Size "19"}
TYPE EL2809_2B6483BD EXTENDS TcoIo.EtcSlaveTerminalBase_947E5A46 :
STRUCT
	{attribute addProperty Name "Channel_1"}
	Channel_1 : Channel_42CA91F7;
	{attribute addProperty Name "Channel_2"}
	Channel_2 : Channel_42CA91F7;
	{attribute addProperty Name "Channel_3"}
	Channel_3 : Channel_42CA91F7;
	{attribute addProperty Name "Channel_4"}
	Channel_4 : Channel_42CA91F7;
	{attribute addProperty Name "Channel_5"}
	Channel_5 : Channel_42CA91F7;
	{attribute addProperty Name "Channel_6"}
	Channel_6 : Channel_42CA91F7;
	{attribute addProperty Name "Channel_7"}
	Channel_7 : Channel_42CA91F7;
	{attribute addProperty Name "Channel_8"}
	Channel_8 : Channel_42CA91F7;
	{attribute addProperty Name "Channel_9"}
	Channel_9 : Channel_42CA91F7;
	{attribute addProperty Name "Channel_10"}
	Channel_10 : Channel_42CA91F7;
	{attribute addProperty Name "Channel_11"}
	Channel_11 : Channel_42CA91F7;
	{attribute addProperty Name "Channel_12"}
	Channel_12 : Channel_42CA91F7;
	{attribute addProperty Name "Channel_13"}
	Channel_13 : Channel_42CA91F7;
	{attribute addProperty Name "Channel_14"}
	Channel_14 : Channel_42CA91F7;
	{attribute addProperty Name "Channel_15"}
	Channel_15 : Channel_42CA91F7;
	{attribute addProperty Name "Channel_16"}
	Channel_16 : Channel_42CA91F7;
	{attribute addProperty Name "WcState"}
	WcState : TcoIo.WcState_0B2B16F9;
	{attribute addProperty Name "InfoData"}
	InfoData : TcoIo.InfoData_6F19DB2B;
END_STRUCT
END_TYPE

// ---- DUTs/IO/Boxes/EL9011_D65D3D32.TcDUT
{attribute 'GeneratedUsingTerminal: EL9011--0000'}
{attribute addProperty VendorId "#x00000002"}
{attribute addProperty BoxType "EL9011--0000"}
{attribute addProperty Description "EL9011 End Terminal"}
{attribute addProperty Physics ""}
{attribute addProperty Id "EL9011"}
{attribute addProperty CRC "3596434738"}
{attribute addProperty Size "0"}
TYPE EL9011_D65D3D32 EXTENDS TcoIo.EtcSlaveEndTerminalBase_866C7F0C :
STRUCT
END_STRUCT
END_TYPE

// ---- DUTs/IO/Devices/SyncUnitTasks_4BE01469.TcDUT
{attribute 'GeneratedUsingTerminal: '}
{attribute addProperty BoxType ""}
{attribute addProperty Id "unreferencedAT %I*SyncUnitTask_AB2F50799PlcTaskAT %I*SyncUnitTask_AB2F50799"}
{attribute addProperty CRC "1272976489"}
{attribute addProperty Size "18"}
TYPE SyncUnitTasks_4BE01469 EXTENDS TcoIo.SyncUnitTasksBase_7C8711EB :
STRUCT
	{attribute addProperty Name "unreferenced"}
	unreferenced : TcoIo.SyncUnitTask_AB2F5079;
	{attribute addProperty Name "PlcTask"}
	PlcTask : TcoIo.SyncUnitTask_AB2F5079;
END_STRUCT
END_TYPE

// ---- DUTs/IO/Devices/SyncUnits_67D36DDA.TcDUT
{attribute 'GeneratedUsingTerminal: '}
{attribute addProperty BoxType ""}
{attribute addProperty Id "_defaultAT %I*SyncUnitTasks_4BE0146918"}
{attribute addProperty CRC "1741909466"}
{attribute addProperty Size "18"}
TYPE SyncUnits_67D36DDA EXTENDS TcoIo.SyncUnitsBase_AD6C35CE :
STRUCT
	{attribute addProperty Name "_default"}
	_default : SyncUnitTasks_4BE01469;
END_STRUCT
END_TYPE

// ---- GVLs/GVL_iXlinker.TcGVL
{attribute 'qualified_only'}
VAR_GLOBAL
		EC1 : EC1_880CB0B9;
		Axis1 : TcoDrivesBeckhoff.TcoAxisRef;
END_VAR

// ---- Abstractions/CUBase/ICUBase.TcIO
INTERFACE ICUBase

PROPERTY AutomatTask : REFERENCE TO CUBaseAutomat
GET
END_GET
END_PROPERTY

PROPERTY GroundTask : REFERENCE TO CUBaseGround
GET
END_GET
END_PROPERTY

PROPERTY  ManualTask : REFERENCE TO TcoTaskedService
GET
END_GET
END_PROPERTY

PROPERTY ProcessDataManager : REFERENCE TO ProcessDataManager
GET
END_GET
END_PROPERTY

PROPERTY RecoverTask : REFERENCE TO CUBaseRecover
GET
END_GET
END_PROPERTY

PROPERTY StatusInfo :REFERENCE TO CuBaseStatusInfo
GET
END_GET
END_PROPERTY

PROPERTY SuspendTask : REFERENCE TO CUBaseSuspend
GET
END_GET
END_PROPERTY

END_INTERFACE

// ---- Abstractions/Safety/ControlButtons/ITcoControlButtons.TcIO
INTERFACE ITcoControlButtons

PROPERTY ButtonAuto : BOOL
GET
END_GET
SET
END_SET
END_PROPERTY

PROPERTY ButtonGround : BOOL
GET
END_GET
SET
END_SET
END_PROPERTY

PROPERTY ButtonRecover : BOOL
GET
END_GET
SET
END_SET
END_PROPERTY

PROPERTY ButtonSuspend : BOOL
GET
END_GET
SET
END_SET
END_PROPERTY

END_INTERFACE

// ---- Abstractions/Safety/ControlVoltage/ITcoControlVoltage.TcIO
INTERFACE ITcoControlVoltage

PROPERTY IsOff : BOOL
GET
END_GET
END_PROPERTY

PROPERTY IsOn : BOOL
GET
END_GET
END_PROPERTY

END_INTERFACE

// ---- Abstractions/Safety/DoorCircuit/ITcoDoorCircuit.TcIO
INTERFACE ITcoDoorCircuit

{attribute 'monitoring' := 'call'}
PROPERTY IsClosed : BOOL
GET
END_GET
END_PROPERTY

{attribute 'monitoring' := 'call'}
PROPERTY IsGlobalVoltageOk : BOOL
GET
END_GET
END_PROPERTY

{attribute 'monitoring' := 'call'}
PROPERTY IsLocalDoorsVoltageOk : BOOL
GET
END_GET
END_PROPERTY

{attribute 'monitoring' := 'call'}
PROPERTY IsLocalVoltageOk : BOOL
GET
END_GET
END_PROPERTY

{attribute 'monitoring' := 'call'}
PROPERTY IsLocked : BOOL
GET
END_GET
END_PROPERTY

{attribute 'monitoring' := 'call'}
PROPERTY IsUnLocked : BOOL
GET
END_GET
END_PROPERTY

METHOD Lock : BOOL
VAR_INPUT
END_VAR
END_METHOD

METHOD UnLock : BOOL
VAR_INPUT
END_VAR
END_METHOD

END_INTERFACE

// ---- Abstractions/Safety/KeyMode/ITcoKeyMode.TcIO
INTERFACE ITcoKeyMode

PROPERTY KeyInAuto : BOOL
GET
END_GET
END_PROPERTY

PROPERTY KeyInManual : BOOL
GET
END_GET
END_PROPERTY

PROPERTY KeyInStep : BOOL
GET
END_GET
END_PROPERTY

END_INTERFACE

// ---- Abstractions/Safety/KeyNormalService/ITcoKeyNormalSevice.TcIO
INTERFACE ITcoKeyNormalSevice

PROPERTY KeyInNormal : BOOL
GET
END_GET
END_PROPERTY

PROPERTY KeyInService : BOOL
GET
END_GET
END_PROPERTY

END_INTERFACE

// ---- Abstractions/Components/MtsFeeding/Blisters/Plb/TcoPlbPaletizator.TcPOU
FUNCTION_BLOCK TcoPlbPaletizator EXTENDS TcoCore.TcoComponent
VAR_INPUT
    inSafeCondition : BOOL;
    inLightCurtainOk : BOOL;
END_VAR

VAR_OUTPUT
END_VAR
VAR
    {attribute addProperty Name "<#Config#>"}
    _config : TcoPlbPaletizator_Config_v_1_x_x;
    {attribute addProperty Name "<#Status#>"}
    {attribute clr [ReadOnly()]}
    _status : TcoPlbPaletizator_Status_v_1_x_x;
    {attribute addProperty Name "<#Control#>"}
    _control : TcoPlbPaletizator_Control_v_1_x_x;

    {attribute addProperty Name "<#Components#>"}
    _components : TcoPlbPaletizator_Components := (Parent := THIS^);

    {attribute addProperty Name "<#Poziadavka novy blister#>"}
    _feedNewBlisterTask : TcoFeedingSequenceTask(THIS^);
    {attribute addProperty Name "<#Poziadavka vylozenie blistera#>"}
    _throwBlisterTask : TcoFeedingSequenceTask(THIS^);

    {attribute addProperty Name "<#Poziadavka vychodzej polohy#>"}
    _setToDefaultTask : TcoFeedingSequenceTask(THIS^);

    {attribute addProperty Name "<#Restore#>"}
    _restoreTask : TcoCore.TcoTask(THIS^);

    {attribute addProperty Name "<#Test positions#>"}
    _positions : TcoPlbPaletizator_Positions(THIS^);

    {attribute clr [CompilerOmits("BuilderPlainer", "BuilderOnliner","BuilderOnlinerInterface","BuilderShadowerInterface")]}
    _blinker : TcoBlinker(THIS^);
    _timerEntryEmpty : ton;
    _timerOutFull : ton;
    _timerDisableSafety : TON;
    {attribute addProperty Name "<#Temporarily disabled safety#>"}
    _temporarilyDisableSafety : BOOL;

    {attribute clr [CompilerOmits("BuilderPlainer", "BuilderOnliner","BuilderOnlinerInterface","BuilderShadowerInterface")]}
    restoreDone : BOOL;
    {attribute clr [CompilerOmits("BuilderPlainer", "BuilderOnliner","BuilderOnlinerInterface","BuilderShadowerInterface")]}
    _setSequencesToStep : BOOL := FALSE;
    _requiredPosition : TcoDrivesBeckhoff.TcoMultiAxisMoveParam;

END_VAR

_status.SafeCondition:=inSafeCondition;

Context.Environment.Messaging.Suspend();
_status.ReadyToUnloadComponents:=
			Components.P1_PositionUnit.AtWork 
			AND Components.I11_BlisterInWorkPosition.Signal
			AND Components.P2_FixUnit.AtWork
			AND (_positions.WorkPos.Axis1.Position-10)< Components.Manipulator.Axis.AxisStatus.ActPos
			AND (_positions.WorkPos.Axis1.Position+10)> Components.Manipulator.Axis.AxisStatus.ActPos ;

_status.OutBufferFull:= (Components.I9_iThrowBuffer1Isfull.Signal AND NOT _config.EmptyBuffer1Disabled )
				XOR  (Components.I10_iThrowBuffer2Isfull.Signal AND NOT _config.EmptyBuffer2Disabled );

_status.EntryBufferEmpty:=NOT ((Components.I1_iBuffer1HasNotCriticalLevel.Signal OR  _config.Buffer1Disabled)
	AND (Components.I3_iBuffer2HasNotCriticalLevel.Signal OR  _config.Buffer2Disabled) 
	AND (Components.I5_iBuffer3HasNotCriticalLevel.Signal OR  _config.Buffer3Disabled)
	AND (Components.I7_iBuffer4HasNotCriticalLevel.Signal OR  _config.Buffer4Disabled));				
Context.Environment.Messaging.Resume();

	
IF _config.StepModeManagableFromOutside THEN
	IF _setSequencesToStep THEN
		_feedNewBlisterTask.SetStepMode();
		_throwBlisterTask.SetStepMode();
		_setToDefaultTask.SetStepMode();
	ELSE 
		_feedNewBlisterTask.SetCyclicMode();
		_throwBlisterTask.SetCyclicMode();
		_setToDefaultTask.SetCyclicMode();
	END_IF
END_IF;

_feedNewBlisterTask.Enabled :=NOT _throwBlisterTask.Busy;
IF(_feedNewBlisterTask.Execute())THEN
	SequenceIncomingBlister(refSequenceTask:=_feedNewBlisterTask );
END_IF;

_throwBlisterTask.Enabled :=NOT _feedNewBlisterTask.Busy;
IF(_throwBlisterTask.Execute())THEN
	SequenceOutgoingBlister(refSequenceTask:=_throwBlisterTask);
END_IF;



_setToDefaultTask.Enabled :=TRUE;
IF(_setToDefaultTask.Execute())THEN
	SequenceSetToDefault(refSequenceTask:=_setToDefaultTask,inResetOnlyManipulator:=_control.ResetOnlyManipulator);
END_IF;


//IF NOT inLightCurtainOk THEN
//	Components.Manipulator.Restore();
//END_IF

//*************RESTORE********************

_restoreTask.Enabled := TRUE;
IF _restoreTask.Execute() THEN
	Restore();
	_restoreTask.DoneWhen(inCondition:=TRUE);
END_IF
//****************************************


//********************SAFETY******************
_timerDisableSafety(IN:=_temporarilyDisableSafety,PT:=_config.TimeToDisableSafety);

THIS^.Messenger.OnCondition(inCondition:=_temporarilyDisableSafety).Warning('SAFTY TEMPORARILY DISABLED!');

IF NOT  _temporarilyDisableSafety THEN
	Components.Manipulator.inEnableNegative:=NOT Components.P1_PositionUnit.AtHome;
	Components.Manipulator.inEnablePositive:=NOT Components.P1_PositionUnit.AtHome;

	
    Components.P1_PositionUnit
        .SuspendMoveWorkExpression( Components.P1_PositionUnit.MoveWorkTask.Busy AND NOT inSafeCondition, '<#Movement is blocked due safe zone is interupted(robot in zone)#>');

    Components.P1_PositionUnit
        .SuspendMoveHomeExpression(Components.P1_PositionUnit.MoveHomeTask.Busy AND NOT inSafeCondition, '<#Movement is blocked due safe zone is interupted(robot in zone)#>');

